LIN {X 0,Y 249.476,Z 395.408,A -85,B 0,C 180,E1 -18908.097,E2 -18908.097} C_VEL
LIN {X 0,Y 249.248,Z 395.426,A -85,B 0,C 180,E1 -18911.384,E2 -18911.384} C_VEL
LIN {X 0,Y 249.214,Z 395.443,A -85,B 0,C 180,E1 -18916.504,E2 -18916.504} C_VEL
LIN {X 0,Y 249.083,Z 395.455,A -85,B 0,C 180,E1 -18921.519,E2 -18921.519} C_VEL
LIN {X 0,Y 249.127,Z 395.443,A -85,B 0,C 180,E1 -18925.483,E2 -18925.483} C_VEL
LIN {X 0,Y 249.08,Z 395.458,A -85,B 0,C 180,E1 -18928.994,E2 -18928.994} C_VEL
LIN {X 0,Y 249.033,Z 395.457,A -85,B 0,C 180,E1 -18932.426,E2 -18932.426} C_VEL
LIN {X 0,Y 249.073,Z 395.454,A -85,B 0,C 180,E1 -18936.338,E2 -18936.338} C_VEL
LIN {X 0,Y 249.075,Z 395.455,A -85,B 0,C 180,E1 -18940.465,E2 -18940.465} C_VEL
LIN {X 0,Y 249.018,Z 395.462,A -85,B 0,C 180,E1 -18944.876,E2 -18944.876} C_VEL
LIN {X 0,Y 249.023,Z 395.464,A -85,B 0,C 180,E1 -18947.366,E2 -18947.366} C_VEL
LIN {X 0,Y 249.038,Z 395.463,A -85,B 0,C 180,E1 -18951.623,E2 -18951.623} C_VEL
LIN {X 0,Y 249.062,Z 395.462,A -85,B 0,C 180,E1 -18955.643,E2 -18955.643} C_VEL
LIN {X 0,Y 249.049,Z 395.473,A -85,B 0,C 180,E1 -18956.512,E2 -18956.512} C_VEL
LIN {X 0,Y 249.154,Z 395.988,A -85,B 0,C 180,E1 -18956.721,E2 -18956.721} C_VEL
LIN {X 0,Y 250.368,Z 398.762,A -85,B 0,C 180,E1 -18956.998,E2 -18956.998} C_VEL
LIN {X 0,Y 253.326,Z 404.095,A -85,B 0,C 180,E1 -18957.613,E2 -18957.613} C_VEL
LIN {X 0,Y 260.759,Z 419.272,A -85,B 0,C 180,E1 -18959.134,E2 -18959.134} C_VEL
LIN {X 0,Y 267.463,Z 435.997,A -85,B 0,C 180,E1 -18960.506,E2 -18960.506} C_VEL
LIN {X 0,Y 265.237,Z 502.126,A -85,B 0,C 180,E1 -18962.276,E2 -18962.276} C_VEL
LIN {X 0,Y 264.22,Z 515.294,A -85,B 0,C 180,E1 -18962.905,E2 -18962.905} C_VEL
LIN {X 0,Y 262.927,Z 527.996,A -85,B 0,C 180,E1 -18963.83,E2 -18963.83} C_VEL
LIN {X 0,Y 261.369,Z 539.299,A -85,B 0,C 180,E1 -18964.945,E2 -18964.945} C_VEL
LIN {X 0,Y 259.357,Z 550.925,A -85,B 0,C 180,E1 -18966.442,E2 -18966.442} C_VEL
LIN {X 0,Y 257.651,Z 559.929,A -85,B 0,C 180,E1 -18967.9,E2 -18967.9} C_VEL
LIN {X 0,Y 255.577,Z 569.881,A -85,B 0,C 180,E1 -18969.896,E2 -18969.896} C_VEL
LIN {X 0,Y 253.7,Z 577.735,A -85,B 0,C 180,E1 -18971.842,E2 -18971.842} C_VEL
LIN {X 0,Y 251.774,Z 585.406,A -85,B 0,C 180,E1 -18974.207,E2 -18974.207} C_VEL
LIN {X 0,Y 249.982,Z 592.445,A -85,B 0,C 180,E1 -18977.003,E2 -18977.003} C_VEL
LIN {X 0,Y 248.812,Z 597.131,A -85,B 0,C 180,E1 -18979.421,E2 -18979.421} C_VEL
LIN {X 0,Y 248.008,Z 600.712,A -85,B 0,C 180,E1 -18981.855,E2 -18981.855} C_VEL
LIN {X 0,Y 247.651,Z 602.56,A -85,B 0,C 180,E1 -18983.482,E2 -18983.482} C_VEL
LIN {X 0,Y 247.401,Z 603.948,A -85,B 0,C 180,E1 -18985.111,E2 -18985.111} C_VEL
LIN {X 0,Y 247.213,Z 604.936,A -85,B 0,C 180,E1 -18986.741,E2 -18986.741} C_VEL
LIN {X 0,Y 247.04,Z 605.774,A -85,B 0,C 180,E1 -18990,E2 -18990} C_VEL
LIN {X 0,Y 247.077,Z 605.581,A -85,B 0,C 180,E1 -18991.63,E2 -18991.63} C_VEL
LIN {X 0,Y 247.213,Z 604.996,A -85,B 0,C 180,E1 -18993.259,E2 -18993.259} C_VEL
LIN {X 0,Y 247.402,Z 604.031,A -85,B 0,C 180,E1 -18994.889,E2 -18994.889} C_VEL
LIN {X 0,Y 247.724,Z 602.386,A -85,B 0,C 180,E1 -18996.801,E2 -18996.801} C_VEL
LIN {X 0,Y 248.485,Z 598.627,A -85,B 0,C 180,E1 -18999.77,E2 -18999.77} C_VEL
LIN {X 0,Y 249.513,Z 594.382,A -85,B 0,C 180,E1 -19002.195,E2 -19002.195} C_VEL
LIN {X 0,Y 251.192,Z 587.949,A -85,B 0,C 180,E1 -19004.999,E2 -19004.999} C_VEL
LIN {X 0,Y 252.884,Z 580.88,A -85,B 0,C 180,E1 -19007.383,E2 -19007.383} C_VEL
LIN {X 0,Y 255.134,Z 572.063,A -85,B 0,C 180,E1 -19009.721,E2 -19009.721} C_VEL
LIN {X 0,Y 257.091,Z 562.672,A -85,B 0,C 180,E1 -19011.732,E2 -19011.732} C_VEL
LIN {X 0,Y 258.977,Z 552.995,A -85,B 0,C 180,E1 -19013.383,E2 -19013.383} C_VEL
LIN {X 0,Y 261.03,Z 541.835,A -85,B 0,C 180,E1 -19014.878,E2 -19014.878} C_VEL
LIN {X 0,Y 262.909,Z 529.302,A -85,B 0,C 180,E1 -19016.172,E2 -19016.172} C_VEL
LIN {X 0,Y 264.228,Z 516.356,A -85,B 0,C 180,E1 -19017.15,E2 -19017.15} C_VEL
LIN {X 0,Y 265.322,Z 503.559,A -85,B 0,C 180,E1 -19017.776,E2 -19017.776} C_VEL
LIN {X 0,Y 265.989,Z 484.214,A -85,B 0,C 180,E1 -19018.344,E2 -19018.344} C_VEL
LIN {X 0,Y 267.501,Z 436.029,A -85,B 0,C 180,E1 -19019.618,E2 -19019.618} C_VEL
LIN {X 0,Y 261.46,Z 420.884,A -85,B 0,C 180,E1 -19020.856,E2 -19020.856} C_VEL
LIN {X 0,Y 254.384,Z 406.189,A -85,B 0,C 180,E1 -19022.303,E2 -19022.303} C_VEL
LIN {X 0,Y 250.5,Z 398.916,A -85,B 0,C 180,E1 -19023.116,E2 -19023.116} C_VEL
LIN {X 0,Y 249.299,Z 396.567,A -85,B 0,C 180,E1 -19023.377,E2 -19023.377} C_VEL
LIN {X 0,Y 249.108,Z 395.797,A -85,B 0,C 180,E1 -19023.482,E2 -19023.482} C_VEL
LIN {X 0,Y 249.054,Z 395.456,A -85,B 0,C 180,E1 -19023.779,E2 -19023.779} C_VEL
LIN {X 0,Y 249.055,Z 395.462,A -85,B 0,C 180,E1 -19027.803,E2 -19027.803} C_VEL
LIN {X 0,Y 249.026,Z 395.464,A -85,B 0,C 180,E1 -19030.473,E2 -19030.473} C_VEL
LIN {X 0,Y 249.017,Z 395.465,A -85,B 0,C 180,E1 -19034.875,E2 -19034.875} C_VEL
LIN {X 0,Y 249.06,Z 395.443,A -85,B 0,C 180,E1 -19037.372,E2 -19037.372} C_VEL
LIN {X 0,Y 249.05,Z 395.46,A -85,B 0,C 180,E1 -19041.623,E2 -19041.623} C_VEL
LIN {X 0,Y 249.058,Z 395.459,A -85,B 0,C 180,E1 -19045.642,E2 -19045.642} C_VEL
LIN {X 0,Y 249.048,Z 395.464,A -85,B 0,C 180,E1 -19049.472,E2 -19049.472} C_VEL
LIN {X 0,Y 249.07,Z 395.458,A -85,B 0,C 180,E1 -19053.162,E2 -19053.162} C_VEL
LIN {X 0,Y 249.075,Z 395.451,A -85,B 0,C 180,E1 -19056.732,E2 -19056.732} C_VEL
LIN {X 0,Y 249.106,Z 395.453,A -85,B 0,C 180,E1 -19060.211,E2 -19060.211} C_VEL
LIN {X 0,Y 249.238,Z 395.433,A -85,B 0,C 180,E1 -19063.621,E2 -19063.621} C_VEL
LIN {X 0,Y 249.248,Z 395.429,A -85,B 0,C 180,E1 -19068.616,E2 -19068.616} C_VEL
LIN {X 0,Y 249.476,Z 395.408,A -85,B 0,C 180,E1 -19071.903,E2 -19071.903} C_VEL
LIN {X 0,Y 249.431,Z 395.408,A -85,B 0,C 180,E1 -19076.769,E2 -19076.769} C_VEL
LIN {X 0,Y 249.73,Z 395.374,A -85,B 0,C 180,E1 -19080,E2 -19080} C_VEL
LIN {X 0,Y 249.432,Z 395.408,A -85,B 0,C 180,E1 -19083.23,E2 -19083.23} C_VEL
LIN {X 0,Y 249.476,Z 395.399,A -85,B 0,C 180,E1 -19088.097,E2 -19088.097} C_VEL
LIN {X 0,Y 249.365,Z 395.418,A -85,B 0,C 180,E1 -19089.868,E2 -19089.868} C_VEL
LIN {X 0,Y 248.589,Z 395.52,A -85,B 0,C 180,E1 -19091.213,E2 -19091.213} C_VEL
LIN {X 0,Y 245.727,Z 395.879,A -85,B 0,C 180,E1 -19093.408,E2 -19093.408} C_VEL
LIN {X 0,Y 242.501,Z 396.283,A -85,B 0,C 180,E1 -19096.112,E2 -19096.112} C_VEL
LIN {X 0,Y 242.128,Z 396.324,A -85,B 0,C 180,E1 -19097.048,E2 -19097.048} C_VEL
LIN {X 0,Y 242.049,Z 396.333,A -85,B 0,C 180,E1 -19101.703,E2 -19101.703} C_VEL
LIN {X 0,Y 242.063,Z 396.329,A -85,B 0,C 180,E1 -19105.839,E2 -19105.839} C_VEL
LIN {X 0,Y 242.027,Z 396.335,A -85,B 0,C 180,E1 -19109.581,E2 -19109.581} C_VEL
LIN {X 0,Y 241.988,Z 396.333,A -85,B 0,C 180,E1 -19113.492,E2 -19113.492} C_VEL
LIN {X 0,Y 242.009,Z 396.332,A -85,B 0,C 180,E1 -19117.578,E2 -19117.578} C_VEL
LIN {X 0,Y 241.982,Z 396.34,A -85,B 0,C 180,E1 -19121.913,E2 -19121.913} C_VEL
LIN {X 0,Y 241.982,Z 396.34,A -85,B 0,C 180,E1 -19126.559,E2 -19126.559} C_VEL
LIN {X 0,Y 242.016,Z 396.398,A -85,B 0,C 180,E1 -19129.567,E2 -19129.567} C_VEL
LIN {X 0,Y 244.29,Z 405.347,A -85,B 0,C 180,E1 -19133.662,E2 -19133.662} C_VEL
LIN {X 0,Y 245.495,Z 411.011,A -85,B 0,C 180,E1 -19136.045,E2 -19136.045} C_VEL
LIN {X 0,Y 253.567,Z 428.776,A -85,B 0,C 180,E1 -19137.836,E2 -19137.836} C_VEL
LIN {X 0,Y 256.47,Z 436.178,A -85,B 0,C 180,E1 -19138.477,E2 -19138.477} C_VEL
LIN {X 0,Y 260.334,Z 462.518,A -85,B 0,C 180,E1 -19139.817,E2 -19139.817} C_VEL
LIN {X 0,Y 259.804,Z 485.166,A -85,B 0,C 180,E1 -19140.456,E2 -19140.456} C_VEL
LIN {X 0,Y 258.526,Z 519.992,A -85,B 0,C 180,E1 -19141.427,E2 -19141.427} C_VEL
LIN {X 0,Y 257.247,Z 533.889,A -85,B 0,C 180,E1 -19142.106,E2 -19142.106} C_VEL
LIN {X 0,Y 255.619,Z 546.328,A -85,B 0,C 180,E1 -19143.022,E2 -19143.022} C_VEL
LIN {X 0,Y 253.783,Z 557.429,A -85,B 0,C 180,E1 -19144.141,E2 -19144.141} C_VEL
LIN {X 0,Y 251.537,Z 569.003,A -85,B 0,C 180,E1 -19145.663,E2 -19145.663} C_VEL
LIN {X 0,Y 249.214,Z 579.428,A -85,B 0,C 180,E1 -19147.404,E2 -19147.404} C_VEL
LIN {X 0,Y 247.163,Z 587.956,A -85,B 0,C 180,E1 -19149.181,E2 -19149.181} C_VEL
LIN {X 0,Y 245.407,Z 596.129,A -85,B 0,C 180,E1 -19151.293,E2 -19151.293} C_VEL
LIN {X 0,Y 243.553,Z 603.536,A -85,B 0,C 180,E1 -19153.66,E2 -19153.66} C_VEL
LIN {X 0,Y 241.706,Z 610.636,A -85,B 0,C 180,E1 -19156.549,E2 -19156.549} C_VEL
LIN {X 0,Y 240.796,Z 615.372,A -85,B 0,C 180,E1 -19159.064,E2 -19159.064} C_VEL
LIN {X 0,Y 240.204,Z 618.994,A -85,B 0,C 180,E1 -19161.588,E2 -19161.588} C_VEL
LIN {X 0,Y 239.951,Z 620.862,A -85,B 0,C 180,E1 -19163.272,E2 -19163.272} C_VEL
LIN {X 0,Y 239.8,Z 622.418,A -85,B 0,C 180,E1 -19165.182,E2 -19165.182} C_VEL
LIN {X 0,Y 239.888,Z 623.885,A -85,B 0,C 180,E1 -19168.321,E2 -19168.321} C_VEL
LIN {X 0,Y 239.958,Z 624.101,A -85,B 0,C 180,E1 -19170,E2 -19170} C_VEL
LIN {X 0,Y 239.888,Z 623.875,A -85,B 0,C 180,E1 -19171.679,E2 -19171.679} C_VEL
LIN {X 0,Y 239.842,Z 622.244,A -85,B 0,C 180,E1 -19175.043,E2 -19175.043} C_VEL
LIN {X 0,Y 239.922,Z 620.829,A -85,B 0,C 180,E1 -19176.729,E2 -19176.729} C_VEL
LIN {X 0,Y 240.364,Z 617.869,A -85,B 0,C 180,E1 -19179.254,E2 -19179.254} C_VEL
LIN {X 0,Y 241.06,Z 613.867,A -85,B 0,C 180,E1 -19181.775,E2 -19181.775} C_VEL
LIN {X 0,Y 242.463,Z 607.725,A -85,B 0,C 180,E1 -19184.692,E2 -19184.692} C_VEL
LIN {X 0,Y 244.088,Z 601.024,A -85,B 0,C 180,E1 -19187.165,E2 -19187.165} C_VEL
LIN {X 0,Y 246.052,Z 593.06,A -85,B 0,C 180,E1 -19189.51,E2 -19189.51} C_VEL
LIN {X 0,Y 248.057,Z 584.199,A -85,B 0,C 180,E1 -19191.611,E2 -19191.611} C_VEL
LIN {X 0,Y 250.51,Z 573.689,A -85,B 0,C 180,E1 -19193.564,E2 -19193.564} C_VEL
LIN {X 0,Y 252.906,Z 561.859,A -85,B 0,C 180,E1 -19195.293,E2 -19195.293} C_VEL
LIN {X 0,Y 254.97,Z 549.944,A -85,B 0,C 180,E1 -19196.609,E2 -19196.609} C_VEL
LIN {X 0,Y 256.694,Z 537.544,A -85,B 0,C 180,E1 -19197.627,E2 -19197.627} C_VEL
LIN {X 0,Y 258.057,Z 524.771,A -85,B 0,C 180,E1 -19198.352,E2 -19198.352} C_VEL
LIN {X 0,Y 258.828,Z 511.246,A -85,B 0,C 180,E1 -19198.813,E2 -19198.813} C_VEL
LIN {X 0,Y 260.387,Z 463.573,A -85,B 0,C 180,E1 -19200.101,E2 -19200.101} C_VEL
LIN {X 0,Y 256.436,Z 436.34,A -85,B 0,C 180,E1 -19201.477,E2 -19201.477} C_VEL
LIN {X 0,Y 252.323,Z 425.825,A -85,B 0,C 180,E1 -19202.39,E2 -19202.39} C_VEL
LIN {X 0,Y 246.241,Z 412.845,A -85,B 0,C 180,E1 -19203.725,E2 -19203.725} C_VEL
LIN {X 0,Y 245.462,Z 410.826,A -85,B 0,C 180,E1 -19203.941,E2 -19203.941} C_VEL
LIN {X 0,Y 243.561,Z 402.34,A -85,B 0,C 180,E1 -19207.623,E2 -19207.623} C_VEL
LIN {X 0,Y 242.015,Z 396.339,A -85,B 0,C 180,E1 -19210.434,E2 -19210.434} C_VEL
LIN {X 0,Y 241.971,Z 396.331,A -85,B 0,C 180,E1 -19214.191,E2 -19214.191} C_VEL
LIN {X 0,Y 241.982,Z 396.341,A -85,B 0,C 180,E1 -19218.087,E2 -19218.087} C_VEL
LIN {X 0,Y 242.009,Z 396.335,A -85,B 0,C 180,E1 -19222.422,E2 -19222.422} C_VEL
LIN {X 0,Y 241.988,Z 396.335,A -85,B 0,C 180,E1 -19226.508,E2 -19226.508} C_VEL
LIN {X 0,Y 242.033,Z 396.33,A -85,B 0,C 180,E1 -19230.587,E2 -19230.587} C_VEL
LIN {X 0,Y 242.064,Z 396.329,A -85,B 0,C 180,E1 -19234.183,E2 -19234.183} C_VEL
LIN {X 0,Y 242.049,Z 396.329,A -85,B 0,C 180,E1 -19238.297,E2 -19238.297} C_VEL
LIN {X 0,Y 242.159,Z 396.309,A -85,B 0,C 180,E1 -19243.278,E2 -19243.278} C_VEL
LIN {X 0,Y 242.181,Z 396.313,A -85,B 0,C 180,E1 -19248.28,E2 -19248.28} C_VEL
LIN {X 0,Y 242.423,Z 396.285,A -85,B 0,C 180,E1 -19251.665,E2 -19251.665} C_VEL
LIN {X 0,Y 242.256,Z 396.304,A -85,B 0,C 180,E1 -19255.007,E2 -19255.007} C_VEL
LIN {X 0,Y 242.632,Z 396.251,A -85,B 0,C 180,E1 -19258.34,E2 -19258.34} C_VEL
LIN {X 0,Y 242.632,Z 396.26,A -85,B 0,C 180,E1 -19261.66,E2 -19261.66} C_VEL
LIN {X 0,Y 242.422,Z 396.281,A -85,B 0,C 180,E1 -19266.755,E2 -19266.755} C_VEL
LIN {X 0,Y 242.31,Z 396.299,A -85,B 0,C 180,E1 -19270.022,E2 -19270.022} C_VEL
LIN {X 0,Y 242.159,Z 396.321,A -85,B 0,C 180,E1 -19275.141,E2 -19275.141} C_VEL
LIN {X 0,Y 242.068,Z 396.321,A -85,B 0,C 180,E1 -19278.625,E2 -19278.625} C_VEL
LIN {X 0,Y 242.009,Z 396.338,A -85,B 0,C 180,E1 -19282.181,E2 -19282.181} C_VEL
LIN {X 0,Y 242.063,Z 396.321,A -85,B 0,C 180,E1 -19285.839,E2 -19285.839} C_VEL
LIN {X 0,Y 242.027,Z 396.336,A -85,B 0,C 180,E1 -19289.581,E2 -19289.581} C_VEL
LIN {X 0,Y 241.988,Z 396.34,A -85,B 0,C 180,E1 -19293.492,E2 -19293.492} C_VEL
LIN {X 0,Y 242.01,Z 396.334,A -85,B 0,C 180,E1 -19297.578,E2 -19297.578} C_VEL
LIN {X 0,Y 241.983,Z 396.338,A -85,B 0,C 180,E1 -19301.913,E2 -19301.913} C_VEL
LIN {X 0,Y 241.941,Z 396.345,A -85,B 0,C 180,E1 -19305.802,E2 -19305.802} C_VEL
LIN {X 0,Y 241.972,Z 396.344,A -85,B 0,C 180,E1 -19310.285,E2 -19310.285} C_VEL
LIN {X 0,Y 242.036,Z 396.34,A -85,B 0,C 180,E1 -19314.498,E2 -19314.498} C_VEL
LIN {X 0,Y 242.04,Z 396.336,A -85,B 0,C 180,E1 -19315.567,E2 -19315.567} C_VEL
LIN {X 0,Y 243.044,Z 399.221,A -85,B 0,C 180,E1 -19315.873,E2 -19315.873} C_VEL
LIN {X 0,Y 244.567,Z 401.612,A -85,B 0,C 180,E1 -19316.2,E2 -19316.2} C_VEL
LIN {X 0,Y 248.946,Z 409.674,A -85,B 0,C 180,E1 -19317.152,E2 -19317.152} C_VEL
LIN {X 0,Y 256.463,Z 425.531,A -85,B 0,C 180,E1 -19318.754,E2 -19318.754} C_VEL
LIN {X 0,Y 261.273,Z 437.838,A -85,B 0,C 180,E1 -19319.784,E2 -19319.784} C_VEL
LIN {X 0,Y 259.019,Z 501.868,A -85,B 0,C 180,E1 -19321.526,E2 -19321.526} C_VEL
LIN {X 0,Y 258.034,Z 514.926,A -85,B 0,C 180,E1 -19322.153,E2 -19322.153} C_VEL
LIN {X 0,Y 256.595,Z 528.27,A -85,B 0,C 180,E1 -19323.133,E2 -19323.133} C_VEL
LIN {X 0,Y 254.954,Z 539.572,A -85,B 0,C 180,E1 -19324.269,E2 -19324.269} C_VEL
LIN {X 0,Y 252.876,Z 551.196,A -85,B 0,C 180,E1 -19325.8,E2 -19325.8} C_VEL
LIN {X 0,Y 250.827,Z 561.583,A -85,B 0,C 180,E1 -19327.548,E2 -19327.548} C_VEL
LIN {X 0,Y 248.929,Z 570.151,A -85,B 0,C 180,E1 -19329.335,E2 -19329.335} C_VEL
LIN {X 0,Y 246.983,Z 578.004,A -85,B 0,C 180,E1 -19331.33,E2 -19331.33} C_VEL
LIN {X 0,Y 244.938,Z 585.675,A -85,B 0,C 180,E1 -19333.755,E2 -19333.755} C_VEL
LIN {X 0,Y 243.069,Z 592.714,A -85,B 0,C 180,E1 -19336.626,E2 -19336.626} C_VEL
LIN {X 0,Y 241.844,Z 597.399,A -85,B 0,C 180,E1 -19339.112,E2 -19339.112} C_VEL
LIN {X 0,Y 240.976,Z 600.98,A -85,B 0,C 180,E1 -19341.615,E2 -19341.615} C_VEL
LIN {X 0,Y 240.601,Z 602.828,A -85,B 0,C 180,E1 -19343.29,E2 -19343.29} C_VEL
LIN {X 0,Y 240.322,Z 604.216,A -85,B 0,C 180,E1 -19344.967,E2 -19344.967} C_VEL
LIN {X 0,Y 240.135,Z 605.203,A -85,B 0,C 180,E1 -19346.644,E2 -19346.644} C_VEL
LIN {X 0,Y 239.97,Z 606.04,A -85,B 0,C 180,E1 -19350,E2 -19350} C_VEL
LIN {X 0,Y 240.01,Z 605.847,A -85,B 0,C 180,E1 -19351.678,E2 -19351.678} C_VEL
LIN {X 0,Y 240.135,Z 605.262,A -85,B 0,C 180,E1 -19353.356,E2 -19353.356} C_VEL
LIN {X 0,Y 240.601,Z 602.945,A -85,B 0,C 180,E1 -19356.71,E2 -19356.71} C_VEL
LIN {X 0,Y 241.256,Z 600.084,A -85,B 0,C 180,E1 -19359.219,E2 -19359.219} C_VEL
LIN {X 0,Y 242.176,Z 596.204,A -85,B 0,C 180,E1 -19361.72,E2 -19361.72} C_VEL
LIN {X 0,Y 243.505,Z 591.193,A -85,B 0,C 180,E1 -19364.201,E2 -19364.201} C_VEL
LIN {X 0,Y 245.132,Z 584.882,A -85,B 0,C 180,E1 -19366.66,E2 -19366.66} C_VEL
LIN {X 0,Y 247.296,Z 576.974,A -85,B 0,C 180,E1 -19369.076,E2 -19369.076} C_VEL
LIN {X 0,Y 249.265,Z 568.914,A -85,B 0,C 180,E1 -19371.068,E2 -19371.068} C_VEL
LIN {X 0,Y 251.291,Z 559.083,A -85,B 0,C 180,E1 -19373.05,E2 -19373.05} C_VEL
LIN {X 0,Y 253.509,Z 548.002,A -85,B 0,C 180,E1 -19374.79,E2 -19374.79} C_VEL
LIN {X 0,Y 255.44,Z 537.132,A -85,B 0,C 180,E1 -19376.117,E2 -19376.117} C_VEL
LIN {X 0,Y 257.092,Z 525.12,A -85,B 0,C 180,E1 -19377.25,E2 -19377.25} C_VEL
LIN {X 0,Y 258.371,Z 512.757,A -85,B 0,C 180,E1 -19378.093,E2 -19378.093} C_VEL
LIN {X 0,Y 259.221,Z 499.909,A -85,B 0,C 180,E1 -19378.655,E2 -19378.655} C_VEL
LIN {X 0,Y 261.323,Z 437.744,A -85,B 0,C 180,E1 -19380.345,E2 -19380.345} C_VEL
LIN {X 0,Y 255.173,Z 422.628,A -85,B 0,C 180,E1 -19381.655,E2 -19381.655} C_VEL
LIN {X 0,Y 247.567,Z 406.884,A -85,B 0,C 180,E1 -19383.292,E2 -19383.292} C_VEL
LIN {X 0,Y 243.555,Z 399.903,A -85,B 0,C 180,E1 -19384.164,E2 -19384.164} C_VEL
LIN {X 0,Y 242.217,Z 397.34,A -85,B 0,C 180,E1 -19384.471,E2 -19384.471} C_VEL
LIN {X 0,Y 242.035,Z 396.333,A -85,B 0,C 180,E1 -19384.561,E2 -19384.561} C_VEL
LIN {X 0,Y 242.007,Z 396.339,A -85,B 0,C 180,E1 -19388.363,E2 -19388.363} C_VEL
LIN {X 0,Y 241.947,Z 396.347,A -85,B 0,C 180,E1 -19391.919,E2 -19391.919} C_VEL
LIN {X 0,Y 241.989,Z 396.325,A -85,B 0,C 180,E1 -19396.556,E2 -19396.556} C_VEL
LIN {X 0,Y 242.006,Z 396.34,A -85,B 0,C 180,E1 -19400.29,E2 -19400.29} C_VEL
LIN {X 0,Y 242.034,Z 396.335,A -85,B 0,C 180,E1 -19404.497,E2 -19404.497} C_VEL
LIN {X 0,Y 241.973,Z 396.343,A -85,B 0,C 180,E1 -19408.479,E2 -19408.479} C_VEL
LIN {X 0,Y 242.005,Z 396.336,A -85,B 0,C 180,E1 -19412.312,E2 -19412.312} C_VEL
LIN {X 0,Y 242.053,Z 396.326,A -85,B 0,C 180,E1 -19416.015,E2 -19416.015} C_VEL
LIN {X 0,Y 242.033,Z 396.337,A -85,B 0,C 180,E1 -19419.607,E2 -19419.607} C_VEL
LIN {X 0,Y 242.159,Z 396.312,A -85,B 0,C 180,E1 -19423.278,E2 -19423.278} C_VEL
LIN {X 0,Y 242.181,Z 396.309,A -85,B 0,C 180,E1 -19428.279,E2 -19428.279} C_VEL
LIN {X 0,Y 242.423,Z 396.288,A -85,B 0,C 180,E1 -19431.665,E2 -19431.665} C_VEL
LIN {X 0,Y 242.255,Z 396.299,A -85,B 0,C 180,E1 -19435.007,E2 -19435.007} C_VEL
LIN {X 0,Y 242.632,Z 396.26,A -85,B 0,C 180,E1 -19438.34,E2 -19438.34} C_VEL
LIN {X 0,Y 242.632,Z 396.249,A -85,B 0,C 180,E1 -19441.66,E2 -19441.66} C_VEL
LIN {X 0,Y 242.428,Z 396.285,A -85,B 0,C 180,E1 -19446.659,E2 -19446.659} C_VEL
LIN {X 0,Y 242.309,Z 396.297,A -85,B 0,C 180,E1 -19450.022,E2 -19450.022} C_VEL
LIN {X 0,Y 242.162,Z 396.314,A -85,B 0,C 180,E1 -19455.141,E2 -19455.141} C_VEL
LIN {X 0,Y 242.128,Z 396.324,A -85,B 0,C 180,E1 -19457.048,E2 -19457.048} C_VEL
LIN {X 0,Y 241.355,Z 396.419,A -85,B 0,C 180,E1 -19458.436,E2 -19458.436} C_VEL
LIN {X 0,Y 238.411,Z 396.781,A -85,B 0,C 180,E1 -19460.699,E2 -19460.699} C_VEL
LIN {X 0,Y 235.998,Z 397.089,A -85,B 0,C 180,E1 -19462.544,E2 -19462.544} C_VEL
LIN {X 0,Y 235.017,Z 397.206,A -85,B 0,C 180,E1 -19463.976,E2 -19463.976} C_VEL
LIN {X 0,Y 234.962,Z 397.21,A -85,B 0,C 180,E1 -19464.461,E2 -19464.461} C_VEL
LIN {X 0,Y 234.948,Z 397.218,A -85,B 0,C 180,E1 -19468.595,E2 -19468.595} C_VEL
LIN {X 0,Y 234.946,Z 397.21,A -85,B 0,C 180,E1 -19473.118,E2 -19473.118} C_VEL
LIN {X 0,Y 234.943,Z 397.211,A -85,B 0,C 180,E1 -19476.746,E2 -19476.746} C_VEL
LIN {X 0,Y 234.942,Z 397.215,A -85,B 0,C 180,E1 -19481.155,E2 -19481.155} C_VEL
LIN {X 0,Y 234.938,Z 397.215,A -85,B 0,C 180,E1 -19484.116,E2 -19484.116} C_VEL
LIN {X 0,Y 234.935,Z 397.218,A -85,B 0,C 180,E1 -19488.406,E2 -19488.406} C_VEL
LIN {X 0,Y 234.96,Z 397.503,A -85,B 0,C 180,E1 -19488.722,E2 -19488.722} C_VEL
LIN {X 0,Y 237.003,Z 405.178,A -85,B 0,C 180,E1 -19492.421,E2 -19492.421} C_VEL
LIN {X 0,Y 238.278,Z 410.734,A -85,B 0,C 180,E1 -19494.869,E2 -19494.869} C_VEL
LIN {X 0,Y 247.21,Z 430.033,A -85,B 0,C 180,E1 -19496.956,E2 -19496.956} C_VEL
LIN {X 0,Y 250.691,Z 438.946,A -85,B 0,C 180,E1 -19497.763,E2 -19497.763} C_VEL
LIN {X 0,Y 254.252,Z 464.097,A -85,B 0,C 180,E1 -19499.075,E2 -19499.075} C_VEL
LIN {X 0,Y 252.326,Z 519.739,A -85,B 0,C 180,E1 -19500.658,E2 -19500.658} C_VEL
LIN {X 0,Y 250.995,Z 533.631,A -85,B 0,C 180,E1 -19501.347,E2 -19501.347} C_VEL
LIN {X 0,Y 249.303,Z 546.066,A -85,B 0,C 180,E1 -19502.281,E2 -19502.281} C_VEL
LIN {X 0,Y 247.413,Z 557.166,A -85,B 0,C 180,E1 -19503.424,E2 -19503.424} C_VEL
LIN {X 0,Y 245.075,Z 568.739,A -85,B 0,C 180,E1 -19504.977,E2 -19504.977} C_VEL
LIN {X 0,Y 242.664,Z 579.164,A -85,B 0,C 180,E1 -19506.759,E2 -19506.759} C_VEL
LIN {X 0,Y 240.515,Z 587.691,A -85,B 0,C 180,E1 -19508.577,E2 -19508.577} C_VEL
LIN {X 0,Y 238.739,Z 595.369,A -85,B 0,C 180,E1 -19510.598,E2 -19510.598} C_VEL
LIN {X 0,Y 236.685,Z 603.268,A -85,B 0,C 180,E1 -19513.172,E2 -19513.172} C_VEL
LIN {X 0,Y 234.781,Z 610.369,A -85,B 0,C 180,E1 -19516.145,E2 -19516.145} C_VEL
LIN {X 0,Y 233.787,Z 615.104,A -85,B 0,C 180,E1 -19518.732,E2 -19518.732} C_VEL
LIN {X 0,Y 233.145,Z 618.726,A -85,B 0,C 180,E1 -19521.331,E2 -19521.331} C_VEL
LIN {X 0,Y 232.888,Z 620.595,A -85,B 0,C 180,E1 -19523.067,E2 -19523.067} C_VEL
LIN {X 0,Y 232.703,Z 622.334,A -85,B 0,C 180,E1 -19525.313,E2 -19525.313} C_VEL
LIN {X 0,Y 232.797,Z 623.618,A -85,B 0,C 180,E1 -19528.27,E2 -19528.27} C_VEL
LIN {X 0,Y 232.888,Z 623.835,A -85,B 0,C 180,E1 -19530,E2 -19530} C_VEL
LIN {X 0,Y 232.797,Z 623.607,A -85,B 0,C 180,E1 -19531.73,E2 -19531.73} C_VEL
LIN {X 0,Y 232.744,Z 621.976,A -85,B 0,C 180,E1 -19535.197,E2 -19535.197} C_VEL
LIN {X 0,Y 232.867,Z 620.561,A -85,B 0,C 180,E1 -19536.934,E2 -19536.934} C_VEL
LIN {X 0,Y 233.312,Z 617.599,A -85,B 0,C 180,E1 -19539.536,E2 -19539.536} C_VEL
LIN {X 0,Y 234.079,Z 613.597,A -85,B 0,C 180,E1 -19542.132,E2 -19542.132} C_VEL
LIN {X 0,Y 235.552,Z 607.455,A -85,B 0,C 180,E1 -19545.133,E2 -19545.133} C_VEL
LIN {X 0,Y 237.294,Z 600.754,A -85,B 0,C 180,E1 -19547.672,E2 -19547.672} C_VEL
LIN {X 0,Y 239.167,Z 593.466,A -85,B 0,C 180,E1 -19549.893,E2 -19549.893} C_VEL
LIN {X 0,Y 241.442,Z 583.928,A -85,B 0,C 180,E1 -19552.235,E2 -19552.235} C_VEL
LIN {X 0,Y 243.99,Z 573.418,A -85,B 0,C 180,E1 -19554.233,E2 -19554.233} C_VEL
LIN {X 0,Y 246.207,Z 563.018,A -85,B 0,C 180,E1 -19555.804,E2 -19555.804} C_VEL
LIN {X 0,Y 248.315,Z 551.613,A -85,B 0,C 180,E1 -19557.153,E2 -19557.153} C_VEL
LIN {X 0,Y 250.085,Z 539.873,A -85,B 0,C 180,E1 -19558.194,E2 -19558.194} C_VEL
LIN {X 0,Y 251.63,Z 526.548,A -85,B 0,C 180,E1 -19559.017,E2 -19559.017} C_VEL
LIN {X 0,Y 252.545,Z 513.512,A -85,B 0,C 180,E1 -19559.518,E2 -19559.518} C_VEL
LIN {X 0,Y 254.225,Z 464.328,A -85,B 0,C 180,E1 -19560.876,E2 -19560.876} C_VEL
LIN {X 0,Y 250.494,Z 438.21,A -85,B 0,C 180,E1 -19562.242,E2 -19562.242} C_VEL
LIN {X 0,Y 244.956,Z 425.063,A -85,B 0,C 180,E1 -19563.504,E2 -19563.504} C_VEL
LIN {X 0,Y 238.248,Z 410.481,A -85,B 0,C 180,E1 -19565.126,E2 -19565.126} C_VEL
LIN {X 0,Y 236.416,Z 402.809,A -85,B 0,C 180,E1 -19568.628,E2 -19568.628} C_VEL
LIN {X 0,Y 234.918,Z 397.22,A -85,B 0,C 180,E1 -19571.448,E2 -19571.448} C_VEL
LIN {X 0,Y 234.934,Z 397.207,A -85,B 0,C 180,E1 -19574.114,E2 -19574.114} C_VEL
LIN {X 0,Y 234.957,Z 397.215,A -85,B 0,C 180,E1 -19578.398,E2 -19578.398} C_VEL
LIN {X 0,Y 234.952,Z 397.219,A -85,B 0,C 180,E1 -19581.085,E2 -19581.085} C_VEL
LIN {X 0,Y 234.957,Z 397.216,A -85,B 0,C 180,E1 -19585.366,E2 -19585.366} C_VEL
LIN {X 0,Y 234.966,Z 397.211,A -85,B 0,C 180,E1 -19590.157,E2 -19590.157} C_VEL
LIN {X 0,Y 234.991,Z 397.211,A -85,B 0,C 180,E1 -19593.793,E2 -19593.793} C_VEL
LIN {X 0,Y 235.007,Z 397.208,A -85,B 0,C 180,E1 -19598.969,E2 -19598.969} C_VEL
LIN {X 0,Y 235.092,Z 397.188,A -85,B 0,C 180,E1 -19603.059,E2 -19603.059} C_VEL
LIN {X 0,Y 235.113,Z 397.193,A -85,B 0,C 180,E1 -19607.922,E2 -19607.922} C_VEL
LIN {X 0,Y 235.372,Z 397.16,A -85,B 0,C 180,E1 -19611.414,E2 -19611.414} C_VEL
LIN {X 0,Y 235.399,Z 397.165,A -85,B 0,C 180,E1 -19613.141,E2 -19613.141} C_VEL
LIN {X 0,Y 235.591,Z 397.128,A -85,B 0,C 180,E1 -19618.291,E2 -19618.291} C_VEL
LIN {X 0,Y 235.591,Z 397.137,A -85,B 0,C 180,E1 -19621.71,E2 -19621.71} C_VEL
LIN {X 0,Y 235.399,Z 397.157,A -85,B 0,C 180,E1 -19626.859,E2 -19626.859} C_VEL
LIN {X 0,Y 235.234,Z 397.179,A -85,B 0,C 180,E1 -19630.327,E2 -19630.327} C_VEL
LIN {X 0,Y 235.108,Z 397.198,A -85,B 0,C 180,E1 -19635.607,E2 -19635.607} C_VEL
LIN {X 0,Y 235.004,Z 397.197,A -85,B 0,C 180,E1 -19639.206,E2 -19639.206} C_VEL
LIN {X 0,Y 234.957,Z 397.218,A -85,B 0,C 180,E1 -19642.883,E2 -19642.883} C_VEL
LIN {X 0,Y 234.966,Z 397.207,A -85,B 0,C 180,E1 -19646.658,E2 -19646.658} C_VEL
LIN {X 0,Y 234.929,Z 397.215,A -85,B 0,C 180,E1 -19650.568,E2 -19650.568} C_VEL
LIN {X 0,Y 234.958,Z 397.218,A -85,B 0,C 180,E1 -19654.634,E2 -19654.634} C_VEL
LIN {X 0,Y 234.965,Z 397.217,A -85,B 0,C 180,E1 -19658.953,E2 -19658.953} C_VEL
LIN {X 0,Y 234.963,Z 397.216,A -85,B 0,C 180,E1 -19663.469,E2 -19663.469} C_VEL
LIN {X 0,Y 234.921,Z 397.224,A -85,B 0,C 180,E1 -19666.523,E2 -19666.523} C_VEL
LIN {X 0,Y 234.954,Z 397.216,A -85,B 0,C 180,E1 -19671.087,E2 -19671.087} C_VEL
LIN {X 0,Y 235.013,Z 397.215,A -85,B 0,C 180,E1 -19674.425,E2 -19674.425} C_VEL
LIN {X 0,Y 236.113,Z 400.261,A -85,B 0,C 180,E1 -19674.751,E2 -19674.751} C_VEL
LIN {X 0,Y 237.479,Z 402.266,A -85,B 0,C 180,E1 -19675.059,E2 -19675.059} C_VEL
LIN {X 0,Y 242.907,Z 411.835,A -85,B 0,C 180,E1 -19676.293,E2 -19676.293} C_VEL
LIN {X 0,Y 250.151,Z 427.078,A -85,B 0,C 180,E1 -19677.914,E2 -19677.914} C_VEL
LIN {X 0,Y 255.067,Z 439.434,A -85,B 0,C 180,E1 -19679.011,E2 -19679.011} C_VEL
LIN {X 0,Y 254.065,Z 468.718,A -85,B 0,C 180,E1 -19679.819,E2 -19679.819} C_VEL
LIN {X 0,Y 252.777,Z 502.806,A -85,B 0,C 180,E1 -19680.787,E2 -19680.787} C_VEL
LIN {X 0,Y 251.689,Z 516.022,A -85,B 0,C 180,E1 -19681.449,E2 -19681.449} C_VEL
LIN {X 0,Y 250.31,Z 528.543,A -85,B 0,C 180,E1 -19682.402,E2 -19682.402} C_VEL
LIN {X 0,Y 248.592,Z 539.844,A -85,B 0,C 180,E1 -19683.56,E2 -19683.56} C_VEL
LIN {X 0,Y 246.425,Z 551.467,A -85,B 0,C 180,E1 -19685.124,E2 -19685.124} C_VEL
LIN {X 0,Y 244.56,Z 560.439,A -85,B 0,C 180,E1 -19686.642,E2 -19686.642} C_VEL
LIN {X 0,Y 242.308,Z 570.421,A -85,B 0,C 180,E1 -19688.743,E2 -19688.743} C_VEL
LIN {X 0,Y 240.281,Z 578.273,A -85,B 0,C 180,E1 -19690.789,E2 -19690.789} C_VEL
LIN {X 0,Y 238.126,Z 585.945,A -85,B 0,C 180,E1 -19693.277,E2 -19693.277} C_VEL
LIN {X 0,Y 236.173,Z 592.983,A -85,B 0,C 180,E1 -19696.228,E2 -19696.228} C_VEL
LIN {X 0,Y 234.867,Z 597.667,A -85,B 0,C 180,E1 -19698.785,E2 -19698.785} C_VEL
LIN {X 0,Y 233.946,Z 601.248,A -85,B 0,C 180,E1 -19701.361,E2 -19701.361} C_VEL
LIN {X 0,Y 233.491,Z 603.336,A -85,B 0,C 180,E1 -19703.361,E2 -19703.361} C_VEL
LIN {X 0,Y 233.058,Z 605.471,A -85,B 0,C 180,E1 -19706.542,E2 -19706.542} C_VEL
LIN {X 0,Y 232.945,Z 606.077,A -85,B 0,C 180,E1 -19708.271,E2 -19708.271} C_VEL
LIN {X 0,Y 232.901,Z 606.306,A -85,B 0,C 180,E1 -19710,E2 -19710} C_VEL
LIN {X 0,Y 232.945,Z 606.113,A -85,B 0,C 180,E1 -19711.729,E2 -19711.729} C_VEL
LIN {X 0,Y 233.058,Z 605.529,A -85,B 0,C 180,E1 -19713.458,E2 -19713.458} C_VEL
LIN {X 0,Y 233.545,Z 603.211,A -85,B 0,C 180,E1 -19716.913,E2 -19716.913} C_VEL
LIN {X 0,Y 234.236,Z 600.351,A -85,B 0,C 180,E1 -19719.498,E2 -19719.498} C_VEL
LIN {X 0,Y 235.239,Z 596.47,A -85,B 0,C 180,E1 -19722.071,E2 -19722.071} C_VEL
LIN {X 0,Y 236.63,Z 591.459,A -85,B 0,C 180,E1 -19724.622,E2 -19724.622} C_VEL
LIN {X 0,Y 238.334,Z 585.147,A -85,B 0,C 180,E1 -19727.15,E2 -19727.15} C_VEL
LIN {X 0,Y 240.593,Z 577.238,A -85,B 0,C 180,E1 -19729.628,E2 -19729.628} C_VEL
LIN {X 0,Y 242.652,Z 569.178,A -85,B 0,C 180,E1 -19731.671,E2 -19731.671} C_VEL
LIN {X 0,Y 244.764,Z 559.347,A -85,B 0,C 180,E1 -19733.702,E2 -19733.702} C_VEL
LIN {X 0,Y 247.101,Z 548.264,A -85,B 0,C 180,E1 -19735.479,E2 -19735.479} C_VEL
LIN {X 0,Y 249.104,Z 537.393,A -85,B 0,C 180,E1 -19736.833,E2 -19736.833} C_VEL
LIN {X 0,Y 250.806,Z 525.379,A -85,B 0,C 180,E1 -19737.992,E2 -19737.992} C_VEL
LIN {X 0,Y 252.147,Z 513.013,A -85,B 0,C 180,E1 -19738.851,E2 -19738.851} C_VEL
LIN {X 0,Y 253.033,Z 500.159,A -85,B 0,C 180,E1 -19739.423,E2 -19739.423} C_VEL
LIN {X 0,Y 255.182,Z 439.559,A -85,B 0,C 180,E1 -19741.105,E2 -19741.105} C_VEL
LIN {X 0,Y 249.579,Z 425.803,A -85,B 0,C 180,E1 -19742.351,E2 -19742.351} C_VEL
LIN {X 0,Y 242.543,Z 411.061,A -85,B 0,C 180,E1 -19743.935,E2 -19743.935} C_VEL
LIN {X 0,Y 236.521,Z 400.814,A -85,B 0,C 180,E1 -19745.306,E2 -19745.306} C_VEL
LIN {X 0,Y 235.154,Z 398.128,A -85,B 0,C 180,E1 -19745.643,E2 -19745.643} C_VEL
LIN {X 0,Y 234.981,Z 397.216,A -85,B 0,C 180,E1 -19745.72,E2 -19745.72} C_VEL
LIN {X 0,Y 234.941,Z 397.22,A -85,B 0,C 180,E1 -19748.944,E2 -19748.944} C_VEL
LIN {X 0,Y 234.921,Z 397.22,A -85,B 0,C 180,E1 -19753.477,E2 -19753.477} C_VEL
LIN {X 0,Y 234.963,Z 397.199,A -85,B 0,C 180,E1 -19756.531,E2 -19756.531} C_VEL
LIN {X 0,Y 234.953,Z 397.219,A -85,B 0,C 180,E1 -19761.085,E2 -19761.085} C_VEL
LIN {X 0,Y 234.958,Z 397.217,A -85,B 0,C 180,E1 -19765.366,E2 -19765.366} C_VEL
LIN {X 0,Y 234.966,Z 397.213,A -85,B 0,C 180,E1 -19770.157,E2 -19770.157} C_VEL
LIN {X 0,Y 234.991,Z 397.214,A -85,B 0,C 180,E1 -19773.793,E2 -19773.793} C_VEL
LIN {X 0,Y 235.007,Z 397.21,A -85,B 0,C 180,E1 -19778.969,E2 -19778.969} C_VEL
LIN {X 0,Y 235.092,Z 397.191,A -85,B 0,C 180,E1 -19783.059,E2 -19783.059} C_VEL
LIN {X 0,Y 235.113,Z 397.19,A -85,B 0,C 180,E1 -19787.922,E2 -19787.922} C_VEL
LIN {X 0,Y 235.372,Z 397.167,A -85,B 0,C 180,E1 -19791.414,E2 -19791.414} C_VEL
LIN {X 0,Y 235.399,Z 397.162,A -85,B 0,C 180,E1 -19793.141,E2 -19793.141} C_VEL
LIN {X 0,Y 235.591,Z 397.137,A -85,B 0,C 180,E1 -19798.29,E2 -19798.29} C_VEL
LIN {X 0,Y 235.592,Z 397.125,A -85,B 0,C 180,E1 -19801.709,E2 -19801.709} C_VEL
LIN {X 0,Y 235.399,Z 397.158,A -85,B 0,C 180,E1 -19806.859,E2 -19806.859} C_VEL
LIN {X 0,Y 235.234,Z 397.179,A -85,B 0,C 180,E1 -19810.327,E2 -19810.327} C_VEL
LIN {X 0,Y 235.109,Z 397.195,A -85,B 0,C 180,E1 -19815.607,E2 -19815.607} C_VEL
LIN {X 0,Y 235.004,Z 397.203,A -85,B 0,C 180,E1 -19819.206,E2 -19819.206} C_VEL
LIN {X 0,Y 234.957,Z 397.217,A -85,B 0,C 180,E1 -19822.883,E2 -19822.883} C_VEL
LIN {X 0,Y 234.962,Z 397.21,A -85,B 0,C 180,E1 -19824.461,E2 -19824.461} C_VEL
LIN {X 0,Y 234.356,Z 397.29,A -85,B 0,C 180,E1 -19825.892,E2 -19825.892} C_VEL
LIN {X 0,Y 232.791,Z 397.49,A -85,B 0,C 180,E1 -19827.297,E2 -19827.297} C_VEL
LIN {X 0,Y 229.026,Z 397.96,A -85,B 0,C 180,E1 -19830.128,E2 -19830.128} C_VEL
LIN {X 0,Y 227.944,Z 398.089,A -85,B 0,C 180,E1 -19831.606,E2 -19831.606} C_VEL
LIN {X 0,Y 227.848,Z 398.096,A -85,B 0,C 180,E1 -19832.108,E2 -19832.108} C_VEL
LIN {X 0,Y 227.906,Z 398.088,A -85,B 0,C 180,E1 -19836.702,E2 -19836.702} C_VEL
LIN {X 0,Y 227.89,Z 398.091,A -85,B 0,C 180,E1 -19840.363,E2 -19840.363} C_VEL
LIN {X 0,Y 227.907,Z 398.091,A -85,B 0,C 180,E1 -19842.72,E2 -19842.72} C_VEL
LIN {X 0,Y 227.883,Z 398.197,A -85,B 0,C 180,E1 -19847.625,E2 -19847.625} C_VEL
LIN {X 0,Y 230.184,Z 406.96,A -85,B 0,C 180,E1 -19852.024,E2 -19852.024} C_VEL
LIN {X 0,Y 230.966,Z 410.19,A -85,B 0,C 180,E1 -19853.558,E2 -19853.558} C_VEL
LIN {X 0,Y 240.745,Z 431.061,A -85,B 0,C 180,E1 -19855.995,E2 -19855.995} C_VEL
LIN {X 0,Y 244.902,Z 441.495,A -85,B 0,C 180,E1 -19857,E2 -19857} C_VEL
LIN {X 0,Y 248.165,Z 465.164,A -85,B 0,C 180,E1 -19858.273,E2 -19858.273} C_VEL
LIN {X 0,Y 246.231,Z 518.855,A -85,B 0,C 180,E1 -19859.825,E2 -19859.825} C_VEL
LIN {X 0,Y 244.982,Z 531.951,A -85,B 0,C 180,E1 -19860.466,E2 -19860.466} C_VEL
LIN {X 0,Y 243.216,Z 544.696,A -85,B 0,C 180,E1 -19861.407,E2 -19861.407} C_VEL
LIN {X 0,Y 241.065,Z 556.903,A -85,B 0,C 180,E1 -19862.667,E2 -19862.667} C_VEL
LIN {X 0,Y 238.646,Z 568.475,A -85,B 0,C 180,E1 -19864.255,E2 -19864.255} C_VEL
LIN {X 0,Y 236.127,Z 578.899,A -85,B 0,C 180,E1 -19866.076,E2 -19866.076} C_VEL
LIN {X 0,Y 233.897,Z 587.425,A -85,B 0,C 180,E1 -19867.94,E2 -19867.94} C_VEL
LIN {X 0,Y 232.017,Z 594.693,A -85,B 0,C 180,E1 -19869.887,E2 -19869.887} C_VEL
LIN {X 0,Y 230.152,Z 601.841,A -85,B 0,C 180,E1 -19872.22,E2 -19872.22} C_VEL
LIN {X 0,Y 228.428,Z 608.279,A -85,B 0,C 180,E1 -19874.84,E2 -19874.84} C_VEL
LIN {X 0,Y 227.087,Z 613.396,A -85,B 0,C 180,E1 -19877.489,E2 -19877.489} C_VEL
LIN {X 0,Y 226.283,Z 617.38,A -85,B 0,C 180,E1 -19880.165,E2 -19880.165} C_VEL
LIN {X 0,Y 225.818,Z 620.328,A -85,B 0,C 180,E1 -19882.849,E2 -19882.849} C_VEL
LIN {X 0,Y 225.605,Z 622.255,A -85,B 0,C 180,E1 -19885.46,E2 -19885.46} C_VEL
LIN {X 0,Y 225.707,Z 623.351,A -85,B 0,C 180,E1 -19888.216,E2 -19888.216} C_VEL
LIN {X 0,Y 225.819,Z 623.569,A -85,B 0,C 180,E1 -19890,E2 -19890} C_VEL
LIN {X 0,Y 225.708,Z 623.34,A -85,B 0,C 180,E1 -19891.784,E2 -19891.784} C_VEL
LIN {X 0,Y 225.671,Z 622.101,A -85,B 0,C 180,E1 -19894.747,E2 -19894.747} C_VEL
LIN {X 0,Y 225.802,Z 620.293,A -85,B 0,C 180,E1 -19897.152,E2 -19897.152} C_VEL
LIN {X 0,Y 226.283,Z 617.33,A -85,B 0,C 180,E1 -19899.835,E2 -19899.835} C_VEL
LIN {X 0,Y 227.084,Z 613.326,A -85,B 0,C 180,E1 -19902.512,E2 -19902.512} C_VEL
LIN {X 0,Y 228.675,Z 607.185,A -85,B 0,C 180,E1 -19905.6,E2 -19905.6} C_VEL
LIN {X 0,Y 230.527,Z 600.485,A -85,B 0,C 180,E1 -19908.209,E2 -19908.209} C_VEL
LIN {X 0,Y 232.815,Z 591.83,A -85,B 0,C 180,E1 -19910.88,E2 -19910.88} C_VEL
LIN {X 0,Y 234.876,Z 583.658,A -85,B 0,C 180,E1 -19912.891,E2 -19912.891} C_VEL
LIN {X 0,Y 237.485,Z 573.145,A -85,B 0,C 180,E1 -19914.942,E2 -19914.942} C_VEL
LIN {X 0,Y 240.123,Z 561.315,A -85,B 0,C 180,E1 -19916.743,E2 -19916.743} C_VEL
LIN {X 0,Y 242.357,Z 549.398,A -85,B 0,C 180,E1 -19918.113,E2 -19918.113} C_VEL
LIN {X 0,Y 244.224,Z 536.995,A -85,B 0,C 180,E1 -19919.17,E2 -19919.17} C_VEL
LIN {X 0,Y 245.695,Z 523.858,A -85,B 0,C 180,E1 -19919.94,E2 -19919.94} C_VEL
LIN {X 0,Y 246.569,Z 509.115,A -85,B 0,C 180,E1 -19920.444,E2 -19920.444} C_VEL
LIN {X 0,Y 248.08,Z 465.032,A -85,B 0,C 180,E1 -19921.695,E2 -19921.695} C_VEL
LIN {X 0,Y 244.685,Z 440.781,A -85,B 0,C 180,E1 -19923.007,E2 -19923.007} C_VEL
LIN {X 0,Y 239.251,Z 427.869,A -85,B 0,C 180,E1 -19924.303,E2 -19924.303} C_VEL
LIN {X 0,Y 232.502,Z 413.601,A -85,B 0,C 180,E1 -19925.963,E2 -19925.963} C_VEL
LIN {X 0,Y 230.934,Z 410.105,A -85,B 0,C 180,E1 -19926.431,E2 -19926.431} C_VEL
LIN {X 0,Y 229.065,Z 402.472,A -85,B 0,C 180,E1 -19930.112,E2 -19930.112} C_VEL
LIN {X 0,Y 227.894,Z 398.095,A -85,B 0,C 180,E1 -19932.412,E2 -19932.412} C_VEL
LIN {X 0,Y 227.907,Z 398.091,A -85,B 0,C 180,E1 -19937.28,E2 -19937.28} C_VEL
LIN {X 0,Y 227.869,Z 398.098,A -85,B 0,C 180,E1 -19941.914,E2 -19941.914} C_VEL
LIN {X 0,Y 227.887,Z 398.091,A -85,B 0,C 180,E1 -19946.373,E2 -19946.373} C_VEL
LIN {X 0,Y 227.916,Z 398.088,A -85,B 0,C 180,E1 -19950.437,E2 -19950.437} C_VEL
LIN {X 0,Y 227.925,Z 398.09,A -85,B 0,C 180,E1 -19954.425,E2 -19954.425} C_VEL
LIN {X 0,Y 227.958,Z 398.084,A -85,B 0,C 180,E1 -19958.287,E2 -19958.287} C_VEL
LIN {X 0,Y 228.03,Z 398.067,A -85,B 0,C 180,E1 -19962.826,E2 -19962.826} C_VEL
LIN {X 0,Y 228.07,Z 398.072,A -85,B 0,C 180,E1 -19967.543,E2 -19967.543} C_VEL
LIN {X 0,Y 228.301,Z 398.037,A -85,B 0,C 180,E1 -19971.146,E2 -19971.146} C_VEL
LIN {X 0,Y 228.35,Z 398.041,A -85,B 0,C 180,E1 -19972.928,E2 -19972.928} C_VEL
LIN {X 0,Y 228.55,Z 398.004,A -85,B 0,C 180,E1 -19978.238,E2 -19978.238} C_VEL
LIN {X 0,Y 228.55,Z 398.014,A -85,B 0,C 180,E1 -19981.762,E2 -19981.762} C_VEL
LIN {X 0,Y 228.35,Z 398.037,A -85,B 0,C 180,E1 -19987.072,E2 -19987.072} C_VEL
LIN {X 0,Y 228.155,Z 398.057,A -85,B 0,C 180,E1 -19990.651,E2 -19990.651} C_VEL
LIN {X 0,Y 228.058,Z 398.071,A -85,B 0,C 180,E1 -19994.273,E2 -19994.273} C_VEL
LIN {X 0,Y 227.999,Z 398.079,A -85,B 0,C 180,E1 -19997.954,E2 -19997.954} C_VEL
LIN {X 0,Y 227.926,Z 398.093,A -85,B 0,C 180,E1 -20002.33,E2 -20002.33} C_VEL
LIN {X 0,Y 227.94,Z 398.081,A -85,B 0,C 180,E1 -20006.603,E2 -20006.603} C_VEL
LIN {X 0,Y 227.906,Z 398.092,A -85,B 0,C 180,E1 -20010.297,E2 -20010.297} C_VEL
LIN {X 0,Y 227.887,Z 398.097,A -85,B 0,C 180,E1 -20013.719,E2 -20013.719} C_VEL
LIN {X 0,Y 227.869,Z 398.097,A -85,B 0,C 180,E1 -20018.086,E2 -20018.086} C_VEL
LIN {X 0,Y 227.907,Z 398.097,A -85,B 0,C 180,E1 -20022.72,E2 -20022.72} C_VEL
LIN {X 0,Y 227.831,Z 398.102,A -85,B 0,C 180,E1 -20027.761,E2 -20027.761} C_VEL
LIN {X 0,Y 227.869,Z 398.102,A -85,B 0,C 180,E1 -20031.915,E2 -20031.915} C_VEL
LIN {X 0,Y 227.925,Z 398.242,A -85,B 0,C 180,E1 -20033.189,E2 -20033.189} C_VEL
LIN {X 0,Y 228.904,Z 400.93,A -85,B 0,C 180,E1 -20033.477,E2 -20033.477} C_VEL
LIN {X 0,Y 230.67,Z 403.491,A -85,B 0,C 180,E1 -20033.902,E2 -20033.902} C_VEL
LIN {X 0,Y 237.571,Z 415.411,A -85,B 0,C 180,E1 -20035.549,E2 -20035.549} C_VEL
LIN {X 0,Y 244.825,Z 430.777,A -85,B 0,C 180,E1 -20037.247,E2 -20037.247} C_VEL
LIN {X 0,Y 249.033,Z 441.412,A -85,B 0,C 180,E1 -20038.23,E2 -20038.23} C_VEL
LIN {X 0,Y 246.658,Z 502.673,A -85,B 0,C 180,E1 -20039.968,E2 -20039.968} C_VEL
LIN {X 0,Y 245.462,Z 516.388,A -85,B 0,C 180,E1 -20040.662,E2 -20040.662} C_VEL
LIN {X 0,Y 244.065,Z 528.817,A -85,B 0,C 180,E1 -20041.633,E2 -20041.633} C_VEL
LIN {X 0,Y 242.271,Z 540.116,A -85,B 0,C 180,E1 -20042.814,E2 -20042.814} C_VEL
LIN {X 0,Y 240.007,Z 551.738,A -85,B 0,C 180,E1 -20044.411,E2 -20044.411} C_VEL
LIN {X 0,Y 238.029,Z 560.869,A -85,B 0,C 180,E1 -20045.996,E2 -20045.996} C_VEL
LIN {X 0,Y 235.715,Z 570.691,A -85,B 0,C 180,E1 -20048.119,E2 -20048.119} C_VEL
LIN {X 0,Y 233.6,Z 578.542,A -85,B 0,C 180,E1 -20050.217,E2 -20050.217} C_VEL
LIN {X 0,Y 231.337,Z 586.214,A -85,B 0,C 180,E1 -20052.771,E2 -20052.771} C_VEL
LIN {X 0,Y 229.295,Z 593.251,A -85,B 0,C 180,E1 -20055.806,E2 -20055.806} C_VEL
LIN {X 0,Y 227.911,Z 597.936,A -85,B 0,C 180,E1 -20058.438,E2 -20058.438} C_VEL
LIN {X 0,Y 226.918,Z 601.517,A -85,B 0,C 180,E1 -20061.092,E2 -20061.092} C_VEL
LIN {X 0,Y 226.392,Z 603.811,A -85,B 0,C 180,E1 -20063.412,E2 -20063.412} C_VEL
LIN {X 0,Y 225.985,Z 605.738,A -85,B 0,C 180,E1 -20066.434,E2 -20066.434} C_VEL
LIN {X 0,Y 225.834,Z 606.572,A -85,B 0,C 180,E1 -20070,E2 -20070} C_VEL
LIN {X 0,Y 225.859,Z 606.379,A -85,B 0,C 180,E1 -20071.783,E2 -20071.783} C_VEL
LIN {X 0,Y 225.984,Z 605.795,A -85,B 0,C 180,E1 -20073.566,E2 -20073.566} C_VEL
LIN {X 0,Y 226.501,Z 603.478,A -85,B 0,C 180,E1 -20077.129,E2 -20077.129} C_VEL
LIN {X 0,Y 227.244,Z 600.617,A -85,B 0,C 180,E1 -20079.793,E2 -20079.793} C_VEL
LIN {X 0,Y 228.289,Z 596.736,A -85,B 0,C 180,E1 -20082.445,E2 -20082.445} C_VEL
LIN {X 0,Y 229.753,Z 591.725,A -85,B 0,C 180,E1 -20085.07,E2 -20085.07} C_VEL
LIN {X 0,Y 231.557,Z 585.412,A -85,B 0,C 180,E1 -20087.668,E2 -20087.668} C_VEL
LIN {X 0,Y 233.911,Z 577.503,A -85,B 0,C 180,E1 -20090.213,E2 -20090.213} C_VEL
LIN {X 0,Y 236.07,Z 569.442,A -85,B 0,C 180,E1 -20092.307,E2 -20092.307} C_VEL
LIN {X 0,Y 238.281,Z 559.61,A -85,B 0,C 180,E1 -20094.388,E2 -20094.388} C_VEL
LIN {X 0,Y 240.724,Z 548.525,A -85,B 0,C 180,E1 -20096.204,E2 -20096.204} C_VEL
LIN {X 0,Y 242.813,Z 537.653,A -85,B 0,C 180,E1 -20097.587,E2 -20097.587} C_VEL
LIN {X 0,Y 244.571,Z 525.638,A -85,B 0,C 180,E1 -20098.771,E2 -20098.771} C_VEL
LIN {X 0,Y 245.952,Z 513.533,A -85,B 0,C 180,E1 -20099.631,E2 -20099.631} C_VEL
LIN {X 0,Y 246.884,Z 499.983,A -85,B 0,C 180,E1 -20100.248,E2 -20100.248} C_VEL
LIN {X 0,Y 249.12,Z 441.451,A -85,B 0,C 180,E1 -20101.895,E2 -20101.895} C_VEL
LIN {X 0,Y 242.664,Z 425.852,A -85,B 0,C 180,E1 -20103.399,E2 -20103.399} C_VEL
LIN {X 0,Y 235.902,Z 412.295,A -85,B 0,C 180,E1 -20104.993,E2 -20104.993} C_VEL
LIN {X 0,Y 229.846,Z 402.159,A -85,B 0,C 180,E1 -20106.452,E2 -20106.452} C_VEL
LIN {X 0,Y 228.304,Z 399.758,A -85,B 0,C 180,E1 -20106.834,E2 -20106.834} C_VEL
LIN {X 0,Y 227.888,Z 398.1,A -85,B 0,C 180,E1 -20106.987,E2 -20106.987} C_VEL
LIN {X 0,Y 227.835,Z 398.103,A -85,B 0,C 180,E1 -20110.374,E2 -20110.374} C_VEL
LIN {X 0,Y 227.849,Z 398.103,A -85,B 0,C 180,E1 -20114.811,E2 -20114.811} C_VEL
LIN {X 0,Y 227.908,Z 398.076,A -85,B 0,C 180,E1 -20117.738,E2 -20117.738} C_VEL
LIN {X 0,Y 227.869,Z 398.095,A -85,B 0,C 180,E1 -20121.914,E2 -20121.914} C_VEL
LIN {X 0,Y 227.887,Z 398.091,A -85,B 0,C 180,E1 -20126.372,E2 -20126.372} C_VEL
LIN {X 0,Y 227.916,Z 398.091,A -85,B 0,C 180,E1 -20130.437,E2 -20130.437} C_VEL
LIN {X 0,Y 227.925,Z 398.093,A -85,B 0,C 180,E1 -20134.425,E2 -20134.425} C_VEL
LIN {X 0,Y 227.958,Z 398.087,A -85,B 0,C 180,E1 -20138.287,E2 -20138.287} C_VEL
LIN {X 0,Y 228.031,Z 398.069,A -85,B 0,C 180,E1 -20142.826,E2 -20142.826} C_VEL
LIN {X 0,Y 228.07,Z 398.069,A -85,B 0,C 180,E1 -20147.543,E2 -20147.543} C_VEL
LIN {X 0,Y 228.301,Z 398.045,A -85,B 0,C 180,E1 -20151.146,E2 -20151.146} C_VEL
LIN {X 0,Y 228.35,Z 398.042,A -85,B 0,C 180,E1 -20152.928,E2 -20152.928} C_VEL
LIN {X 0,Y 228.55,Z 398.014,A -85,B 0,C 180,E1 -20158.238,E2 -20158.238} C_VEL
LIN {X 0,Y 228.55,Z 398.001,A -85,B 0,C 180,E1 -20161.762,E2 -20161.762} C_VEL
LIN {X 0,Y 228.35,Z 398.033,A -85,B 0,C 180,E1 -20167.072,E2 -20167.072} C_VEL
LIN {X 0,Y 228.159,Z 398.062,A -85,B 0,C 180,E1 -20170.651,E2 -20170.651} C_VEL
LIN {X 0,Y 228.06,Z 398.066,A -85,B 0,C 180,E1 -20174.272,E2 -20174.272} C_VEL
LIN {X 0,Y 227.999,Z 398.082,A -85,B 0,C 180,E1 -20177.954,E2 -20177.954} C_VEL
LIN {X 0,Y 227.926,Z 398.094,A -85,B 0,C 180,E1 -20182.33,E2 -20182.33} C_VEL
LIN {X 0,Y 227.939,Z 398.092,A -85,B 0,C 180,E1 -20186.603,E2 -20186.603} C_VEL
LIN {X 0,Y 227.905,Z 398.094,A -85,B 0,C 180,E1 -20190.297,E2 -20190.297} C_VEL
LIN {X 0,Y 227.848,Z 398.096,A -85,B 0,C 180,E1 -20192.108,E2 -20192.108} C_VEL
LIN {X 0,Y 227.164,Z 398.179,A -85,B 0,C 180,E1 -20193.584,E2 -20193.584} C_VEL
LIN {X 0,Y 224.331,Z 398.537,A -85,B 0,C 180,E1 -20195.995,E2 -20195.995} C_VEL
LIN {X 0,Y 221.941,Z 398.837,A -85,B 0,C 180,E1 -20197.962,E2 -20197.962} C_VEL
LIN {X 0,Y 220.926,Z 398.961,A -85,B 0,C 180,E1 -20199.488,E2 -20199.488} C_VEL
LIN {X 0,Y 220.848,Z 398.968,A -85,B 0,C 180,E1 -20200.005,E2 -20200.005} C_VEL
LIN {X 0,Y 220.83,Z 398.974,A -85,B 0,C 180,E1 -20204.44,E2 -20204.44} C_VEL
LIN {X 0,Y 220.828,Z 399.085,A -85,B 0,C 180,E1 -20206.532,E2 -20206.532} C_VEL
LIN {X 0,Y 223.058,Z 407.416,A -85,B 0,C 180,E1 -20210.94,E2 -20210.94} C_VEL
LIN {X 0,Y 223.737,Z 410.094,A -85,B 0,C 180,E1 -20212.204,E2 -20212.204} C_VEL
LIN {X 0,Y 231.223,Z 425.414,A -85,B 0,C 180,E1 -20214.192,E2 -20214.192} C_VEL
LIN {X 0,Y 237.41,Z 439.419,A -85,B 0,C 180,E1 -20215.755,E2 -20215.755} C_VEL
LIN {X 0,Y 239.143,Z 443.988,A -85,B 0,C 180,E1 -20216.196,E2 -20216.196} C_VEL
LIN {X 0,Y 242.148,Z 466.227,A -85,B 0,C 180,E1 -20217.434,E2 -20217.434} C_VEL
LIN {X 0,Y 240.079,Z 519.147,A -85,B 0,C 180,E1 -20218.997,E2 -20218.997} C_VEL
LIN {X 0,Y 238.729,Z 532.53,A -85,B 0,C 180,E1 -20219.679,E2 -20219.679} C_VEL
LIN {X 0,Y 236.831,Z 545.545,A -85,B 0,C 180,E1 -20220.684,E2 -20220.684} C_VEL
LIN {X 0,Y 234.456,Z 558.226,A -85,B 0,C 180,E1 -20222.072,E2 -20222.072} C_VEL
LIN {X 0,Y 231.98,Z 569.508,A -85,B 0,C 180,E1 -20223.7,E2 -20223.7} C_VEL
LIN {X 0,Y 229.362,Z 579.671,A -85,B 0,C 180,E1 -20225.566,E2 -20225.566} C_VEL
LIN {X 0,Y 226.843,Z 588.833,A -85,B 0,C 180,E1 -20227.696,E2 -20227.696} C_VEL
LIN {X 0,Y 224.869,Z 596.417,A -85,B 0,C 180,E1 -20229.892,E2 -20229.892} C_VEL
LIN {X 0,Y 222.741,Z 603.858,A -85,B 0,C 180,E1 -20232.558,E2 -20232.558} C_VEL
LIN {X 0,Y 220.987,Z 609.836,A -85,B 0,C 180,E1 -20235.261,E2 -20235.261} C_VEL
LIN {X 0,Y 219.787,Z 614.568,A -85,B 0,C 180,E1 -20238.004,E2 -20238.004} C_VEL
LIN {X 0,Y 219.056,Z 618.191,A -85,B 0,C 180,E1 -20240.769,E2 -20240.769} C_VEL
LIN {X 0,Y 218.754,Z 620.06,A -85,B 0,C 180,E1 -20242.617,E2 -20242.617} C_VEL
LIN {X 0,Y 218.52,Z 622.138,A -85,B 0,C 180,E1 -20245.574,E2 -20245.574} C_VEL
LIN {X 0,Y 218.62,Z 623.084,A -85,B 0,C 180,E1 -20248.158,E2 -20248.158} C_VEL
LIN {X 0,Y 218.728,Z 623.302,A -85,B 0,C 180,E1 -20250,E2 -20250} C_VEL
LIN {X 0,Y 218.621,Z 623.073,A -85,B 0,C 180,E1 -20251.842,E2 -20251.842} C_VEL
LIN {X 0,Y 218.571,Z 621.439,A -85,B 0,C 180,E1 -20255.535,E2 -20255.535} C_VEL
LIN {X 0,Y 218.726,Z 620.024,A -85,B 0,C 180,E1 -20257.384,E2 -20257.384} C_VEL
LIN {X 0,Y 219.272,Z 617.061,A -85,B 0,C 180,E1 -20260.153,E2 -20260.153} C_VEL
LIN {X 0,Y 220.104,Z 613.056,A -85,B 0,C 180,E1 -20262.915,E2 -20262.915} C_VEL
LIN {X 0,Y 221.826,Z 606.915,A -85,B 0,C 180,E1 -20266.094,E2 -20266.094} C_VEL
LIN {X 0,Y 223.786,Z 600.216,A -85,B 0,C 180,E1 -20268.778,E2 -20268.778} C_VEL
LIN {X 0,Y 226.101,Z 591.733,A -85,B 0,C 180,E1 -20271.476,E2 -20271.476} C_VEL
LIN {X 0,Y 228.322,Z 583.387,A -85,B 0,C 180,E1 -20273.587,E2 -20273.587} C_VEL
LIN {X 0,Y 231.065,Z 572.874,A -85,B 0,C 180,E1 -20275.684,E2 -20275.684} C_VEL
LIN {X 0,Y 233.811,Z 561.043,A -85,B 0,C 180,E1 -20277.525,E2 -20277.525} C_VEL
LIN {X 0,Y 236.114,Z 549.124,A -85,B 0,C 180,E1 -20278.926,E2 -20278.926} C_VEL
LIN {X 0,Y 238.048,Z 536.72,A -85,B 0,C 180,E1 -20280.003,E2 -20280.003} C_VEL
LIN {X 0,Y 239.536,Z 523.946,A -85,B 0,C 180,E1 -20280.77,E2 -20280.77} C_VEL
LIN {X 0,Y 240.428,Z 509.939,A -85,B 0,C 180,E1 -20281.27,E2 -20281.27} C_VEL
LIN {X 0,Y 242.042,Z 466.058,A -85,B 0,C 180,E1 -20282.537,E2 -20282.537} C_VEL
LIN {X 0,Y 238.904,Z 443.222,A -85,B 0,C 180,E1 -20283.816,E2 -20283.816} C_VEL
LIN {X 0,Y 233.113,Z 429.56,A -85,B 0,C 180,E1 -20285.266,E2 -20285.266} C_VEL
LIN {X 0,Y 226.962,Z 416.675,A -85,B 0,C 180,E1 -20286.855,E2 -20286.855} C_VEL
LIN {X 0,Y 223.673,Z 409.841,A -85,B 0,C 180,E1 -20287.785,E2 -20287.785} C_VEL
LIN {X 0,Y 221.645,Z 402.124,A -85,B 0,C 180,E1 -20291.748,E2 -20291.748} C_VEL
LIN {X 0,Y 220.817,Z 398.97,A -85,B 0,C 180,E1 -20293.48,E2 -20293.48} C_VEL
LIN {X 0,Y 220.851,Z 398.974,A -85,B 0,C 180,E1 -20298.066,E2 -20298.066} C_VEL
LIN {X 0,Y 220.836,Z 398.971,A -85,B 0,C 180,E1 -20302.711,E2 -20302.711} C_VEL
LIN {X 0,Y 220.821,Z 398.971,A -85,B 0,C 180,E1 -20307.245,E2 -20307.245} C_VEL
LIN {X 0,Y 220.833,Z 398.965,A -85,B 0,C 180,E1 -20311.486,E2 -20311.486} C_VEL
LIN {X 0,Y 220.864,Z 398.963,A -85,B 0,C 180,E1 -20315.565,E2 -20315.565} C_VEL
LIN {X 0,Y 220.888,Z 398.97,A -85,B 0,C 180,E1 -20319.514,E2 -20319.514} C_VEL
LIN {X 0,Y 221.012,Z 398.941,A -85,B 0,C 180,E1 -20323.37,E2 -20323.37} C_VEL
LIN {X 0,Y 221.102,Z 398.929,A -85,B 0,C 180,E1 -20329.005,E2 -20329.005} C_VEL
LIN {X 0,Y 221.285,Z 398.919,A -85,B 0,C 180,E1 -20332.701,E2 -20332.701} C_VEL
LIN {X 0,Y 221.508,Z 398.881,A -85,B 0,C 180,E1 -20338.182,E2 -20338.182} C_VEL
LIN {X 0,Y 221.508,Z 398.891,A -85,B 0,C 180,E1 -20341.818,E2 -20341.818} C_VEL
LIN {X 0,Y 221.301,Z 398.917,A -85,B 0,C 180,E1 -20347.298,E2 -20347.298} C_VEL
LIN {X 0,Y 221.102,Z 398.932,A -85,B 0,C 180,E1 -20350.995,E2 -20350.995} C_VEL
LIN {X 0,Y 221.012,Z 398.955,A -85,B 0,C 180,E1 -20356.63,E2 -20356.63} C_VEL
LIN {X 0,Y 220.888,Z 398.958,A -85,B 0,C 180,E1 -20360.487,E2 -20360.487} C_VEL
LIN {X 0,Y 220.864,Z 398.967,A -85,B 0,C 180,E1 -20364.436,E2 -20364.436} C_VEL
LIN {X 0,Y 220.834,Z 398.977,A -85,B 0,C 180,E1 -20368.514,E2 -20368.514} C_VEL
LIN {X 0,Y 220.822,Z 398.971,A -85,B 0,C 180,E1 -20372.756,E2 -20372.756} C_VEL
LIN {X 0,Y 220.836,Z 398.969,A -85,B 0,C 180,E1 -20377.289,E2 -20377.289} C_VEL
LIN {X 0,Y 220.851,Z 398.97,A -85,B 0,C 180,E1 -20381.934,E2 -20381.934} C_VEL
LIN {X 0,Y 220.788,Z 398.979,A -85,B 0,C 180,E1 -20385.551,E2 -20385.551} C_VEL
LIN {X 0,Y 220.809,Z 398.978,A -85,B 0,C 180,E1 -20390.465,E2 -20390.465} C_VEL
LIN {X 0,Y 220.843,Z 398.976,A -85,B 0,C 180,E1 -20391.793,E2 -20391.793} C_VEL
LIN {X 0,Y 221.856,Z 401.875,A -85,B 0,C 180,E1 -20392.141,E2 -20392.141} C_VEL
LIN {X 0,Y 223.504,Z 404.074,A -85,B 0,C 180,E1 -20392.559,E2 -20392.559} C_VEL
LIN {X 0,Y 230.678,Z 416.044,A -85,B 0,C 180,E1 -20394.377,E2 -20394.377} C_VEL
LIN {X 0,Y 237.05,Z 428.891,A -85,B 0,C 180,E1 -20395.948,E2 -20395.948} C_VEL
LIN {X 0,Y 242.465,Z 441.813,A -85,B 0,C 180,E1 -20397.266,E2 -20397.266} C_VEL
LIN {X 0,Y 242.942,Z 443.202,A -85,B 0,C 180,E1 -20397.387,E2 -20397.387} C_VEL
LIN {X 0,Y 240.487,Z 503.645,A -85,B 0,C 180,E1 -20399.151,E2 -20399.151} C_VEL
LIN {X 0,Y 239.219,Z 517.421,A -85,B 0,C 180,E1 -20399.878,E2 -20399.878} C_VEL
LIN {X 0,Y 237.687,Z 530.177,A -85,B 0,C 180,E1 -20400.921,E2 -20400.921} C_VEL
LIN {X 0,Y 235.702,Z 541.968,A -85,B 0,C 180,E1 -20402.233,E2 -20402.233} C_VEL
LIN {X 0,Y 233.357,Z 553.295,A -85,B 0,C 180,E1 -20403.867,E2 -20403.867} C_VEL
LIN {X 0,Y 231.06,Z 563.345,A -85,B 0,C 180,E1 -20405.722,E2 -20405.722} C_VEL
LIN {X 0,Y 228.702,Z 572.646,A -85,B 0,C 180,E1 -20407.887,E2 -20407.887} C_VEL
LIN {X 0,Y 226.068,Z 581.543,A -85,B 0,C 180,E1 -20410.477,E2 -20410.477} C_VEL
LIN {X 0,Y 223.955,Z 588.696,A -85,B 0,C 180,E1 -20413.126,E2 -20413.126} C_VEL
LIN {X 0,Y 222.416,Z 593.52,A -85,B 0,C 180,E1 -20415.358,E2 -20415.358} C_VEL
LIN {X 0,Y 220.976,Z 598.203,A -85,B 0,C 180,E1 -20418.07,E2 -20418.07} C_VEL
LIN {X 0,Y 219.919,Z 601.785,A -85,B 0,C 180,E1 -20420.806,E2 -20420.806} C_VEL
LIN {X 0,Y 219.294,Z 604.287,A -85,B 0,C 180,E1 -20423.465,E2 -20423.465} C_VEL
LIN {X 0,Y 218.913,Z 606.005,A -85,B 0,C 180,E1 -20426.319,E2 -20426.319} C_VEL
LIN {X 0,Y 218.746,Z 606.839,A -85,B 0,C 180,E1 -20430,E2 -20430} C_VEL
LIN {X 0,Y 218.775,Z 606.646,A -85,B 0,C 180,E1 -20431.841,E2 -20431.841} C_VEL
LIN {X 0,Y 218.913,Z 606.061,A -85,B 0,C 180,E1 -20433.681,E2 -20433.681} C_VEL
LIN {X 0,Y 219.472,Z 603.744,A -85,B 0,C 180,E1 -20437.359,E2 -20437.359} C_VEL
LIN {X 0,Y 220.236,Z 600.884,A -85,B 0,C 180,E1 -20440.108,E2 -20440.108} C_VEL
LIN {X 0,Y 221.357,Z 597.002,A -85,B 0,C 180,E1 -20442.841,E2 -20442.841} C_VEL
LIN {X 0,Y 222.899,Z 591.991,A -85,B 0,C 180,E1 -20445.545,E2 -20445.545} C_VEL
LIN {X 0,Y 224.805,Z 585.677,A -85,B 0,C 180,E1 -20448.217,E2 -20448.217} C_VEL
LIN {X 0,Y 227.27,Z 577.768,A -85,B 0,C 180,E1 -20450.831,E2 -20450.831} C_VEL
LIN {X 0,Y 229.493,Z 569.782,A -85,B 0,C 180,E1 -20452.962,E2 -20452.962} C_VEL
LIN {X 0,Y 231.851,Z 559.873,A -85,B 0,C 180,E1 -20455.111,E2 -20455.111} C_VEL
LIN {X 0,Y 234.385,Z 548.787,A -85,B 0,C 180,E1 -20456.969,E2 -20456.969} C_VEL
LIN {X 0,Y 236.568,Z 537.913,A -85,B 0,C 180,E1 -20458.38,E2 -20458.38} C_VEL
LIN {X 0,Y 238.384,Z 525.897,A -85,B 0,C 180,E1 -20459.591,E2 -20459.591} C_VEL
LIN {X 0,Y 239.793,Z 514.031,A -85,B 0,C 180,E1 -20460.453,E2 -20460.453} C_VEL
LIN {X 0,Y 240.733,Z 501.257,A -85,B 0,C 180,E1 -20461.064,E2 -20461.064} C_VEL
LIN {X 0,Y 243.074,Z 443.311,A -85,B 0,C 180,E1 -20462.731,E2 -20462.731} C_VEL
LIN {X 0,Y 236.797,Z 428.207,A -85,B 0,C 180,E1 -20464.264,E2 -20464.264} C_VEL
LIN {X 0,Y 230.885,Z 416.381,A -85,B 0,C 180,E1 -20465.723,E2 -20465.723} C_VEL
LIN {X 0,Y 225.16,Z 406.81,A -85,B 0,C 180,E1 -20467.163,E2 -20467.163} C_VEL
LIN {X 0,Y 222.67,Z 402.934,A -85,B 0,C 180,E1 -20467.81,E2 -20467.81} C_VEL
LIN {X 0,Y 221.136,Z 400.316,A -85,B 0,C 180,E1 -20468.228,E2 -20468.228} C_VEL
LIN {X 0,Y 220.809,Z 398.979,A -85,B 0,C 180,E1 -20468.385,E2 -20468.385} C_VEL
LIN {X 0,Y 220.795,Z 398.978,A -85,B 0,C 180,E1 -20472.937,E2 -20472.937} C_VEL
LIN {X 0,Y 220.865,Z 398.951,A -85,B 0,C 180,E1 -20477.042,E2 -20477.042} C_VEL
LIN {X 0,Y 220.854,Z 398.974,A -85,B 0,C 180,E1 -20480.473,E2 -20480.473} C_VEL
LIN {X 0,Y 220.813,Z 398.98,A -85,B 0,C 180,E1 -20485.047,E2 -20485.047} C_VEL
LIN {X 0,Y 220.865,Z 398.974,A -85,B 0,C 180,E1 -20489.394,E2 -20489.394} C_VEL
LIN {X 0,Y 220.892,Z 398.97,A -85,B 0,C 180,E1 -20493.549,E2 -20493.549} C_VEL
LIN {X 0,Y 220.874,Z 398.964,A -85,B 0,C 180,E1 -20497.553,E2 -20497.553} C_VEL
LIN {X 0,Y 220.98,Z 398.946,A -85,B 0,C 180,E1 -20502.571,E2 -20502.571} C_VEL
LIN {X 0,Y 221.008,Z 398.951,A -85,B 0,C 180,E1 -20507.138,E2 -20507.138} C_VEL
LIN {X 0,Y 221.232,Z 398.923,A -85,B 0,C 180,E1 -20510.86,E2 -20510.86} C_VEL
LIN {X 0,Y 221.285,Z 398.921,A -85,B 0,C 180,E1 -20512.701,E2 -20512.701} C_VEL
LIN {X 0,Y 221.508,Z 398.892,A -85,B 0,C 180,E1 -20518.182,E2 -20518.182} C_VEL
LIN {X 0,Y 221.508,Z 398.878,A -85,B 0,C 180,E1 -20521.818,E2 -20521.818} C_VEL
LIN {X 0,Y 221.285,Z 398.911,A -85,B 0,C 180,E1 -20527.298,E2 -20527.298} C_VEL
LIN {X 0,Y 221.108,Z 398.942,A -85,B 0,C 180,E1 -20530.994,E2 -20530.994} C_VEL
LIN {X 0,Y 221.012,Z 398.953,A -85,B 0,C 180,E1 -20536.63,E2 -20536.63} C_VEL
LIN {X 0,Y 220.888,Z 398.961,A -85,B 0,C 180,E1 -20540.487,E2 -20540.487} C_VEL
LIN {X 0,Y 220.864,Z 398.966,A -85,B 0,C 180,E1 -20544.435,E2 -20544.435} C_VEL
LIN {X 0,Y 220.833,Z 398.976,A -85,B 0,C 180,E1 -20548.514,E2 -20548.514} C_VEL
LIN {X 0,Y 220.821,Z 398.97,A -85,B 0,C 180,E1 -20552.755,E2 -20552.755} C_VEL
LIN {X 0,Y 220.836,Z 398.967,A -85,B 0,C 180,E1 -20557.289,E2 -20557.289} C_VEL
LIN {X 0,Y 220.848,Z 398.968,A -85,B 0,C 180,E1 -20560.005,E2 -20560.005} C_VEL
LIN {X 0,Y 220.201,Z 399.076,A -85,B 0,C 180,E1 -20561.019,E2 -20561.019} C_VEL
LIN {X 0,Y 217.444,Z 399.395,A -85,B 0,C 180,E1 -20562.619,E2 -20562.619} C_VEL
LIN {X 0,Y 214.575,Z 399.752,A -85,B 0,C 180,E1 -20564.251,E2 -20564.251} C_VEL
LIN {X 0,Y 213.795,Z 399.873,A -85,B 0,C 180,E1 -20565.301,E2 -20565.301} C_VEL
LIN {X 0,Y 216,Z 408.337,A -85,B 0,C 180,E1 -20570.009,E2 -20570.009} C_VEL
LIN {X 0,Y 216.444,Z 409.836,A -85,B 0,C 180,E1 -20570.694,E2 -20570.694} C_VEL
LIN {X 0,Y 218.711,Z 414.124,A -85,B 0,C 180,E1 -20571.35,E2 -20571.35} C_VEL
LIN {X 0,Y 225.105,Z 426.982,A -85,B 0,C 180,E1 -20573.132,E2 -20573.132} C_VEL
LIN {X 0,Y 232.157,Z 443.064,A -85,B 0,C 180,E1 -20575.01,E2 -20575.01} C_VEL
LIN {X 0,Y 233.513,Z 446.948,A -85,B 0,C 180,E1 -20575.382,E2 -20575.382} C_VEL
LIN {X 0,Y 236.115,Z 466.566,A -85,B 0,C 180,E1 -20576.515,E2 -20576.515} C_VEL
LIN {X 0,Y 233.977,Z 519.419,A -85,B 0,C 180,E1 -20578.123,E2 -20578.123} C_VEL
LIN {X 0,Y 232.513,Z 533.069,A -85,B 0,C 180,E1 -20578.845,E2 -20578.845} C_VEL
LIN {X 0,Y 230.662,Z 545.284,A -85,B 0,C 180,E1 -20579.82,E2 -20579.82} C_VEL
LIN {X 0,Y 228.187,Z 557.962,A -85,B 0,C 180,E1 -20581.234,E2 -20581.234} C_VEL
LIN {X 0,Y 225.601,Z 569.243,A -85,B 0,C 180,E1 -20582.897,E2 -20582.897} C_VEL
LIN {X 0,Y 222.925,Z 579.407,A -85,B 0,C 180,E1 -20584.812,E2 -20584.812} C_VEL
LIN {X 0,Y 220.254,Z 588.567,A -85,B 0,C 180,E1 -20586.991,E2 -20586.991} C_VEL
LIN {X 0,Y 218.147,Z 596.149,A -85,B 0,C 180,E1 -20589.245,E2 -20589.245} C_VEL
LIN {X 0,Y 215.911,Z 603.59,A -85,B 0,C 180,E1 -20591.988,E2 -20591.988} C_VEL
LIN {X 0,Y 214.111,Z 609.57,A -85,B 0,C 180,E1 -20594.776,E2 -20594.776} C_VEL
LIN {X 0,Y 212.811,Z 614.301,A -85,B 0,C 180,E1 -20597.605,E2 -20597.605} C_VEL
LIN {X 0,Y 212.031,Z 617.924,A -85,B 0,C 180,E1 -20600.461,E2 -20600.461} C_VEL
LIN {X 0,Y 211.68,Z 619.792,A -85,B 0,C 180,E1 -20602.369,E2 -20602.369} C_VEL
LIN {X 0,Y 211.42,Z 622.016,A -85,B 0,C 180,E1 -20605.759,E2 -20605.759} C_VEL
LIN {X 0,Y 211.514,Z 622.817,A -85,B 0,C 180,E1 -20608.096,E2 -20608.096} C_VEL
LIN {X 0,Y 211.64,Z 623.035,A -85,B 0,C 180,E1 -20610,E2 -20610} C_VEL
LIN {X 0,Y 211.516,Z 622.806,A -85,B 0,C 180,E1 -20611.904,E2 -20611.904} C_VEL
LIN {X 0,Y 211.473,Z 621.917,A -85,B 0,C 180,E1 -20614.434,E2 -20614.434} C_VEL
LIN {X 0,Y 211.659,Z 619.755,A -85,B 0,C 180,E1 -20617.632,E2 -20617.632} C_VEL
LIN {X 0,Y 212.239,Z 616.792,A -85,B 0,C 180,E1 -20620.493,E2 -20620.493} C_VEL
LIN {X 0,Y 213.143,Z 612.786,A -85,B 0,C 180,E1 -20623.345,E2 -20623.345} C_VEL
LIN {X 0,Y 215.002,Z 606.646,A -85,B 0,C 180,E1 -20626.619,E2 -20626.619} C_VEL
LIN {X 0,Y 217.067,Z 599.946,A -85,B 0,C 180,E1 -20629.382,E2 -20629.382} C_VEL
LIN {X 0,Y 219.408,Z 591.629,A -85,B 0,C 180,E1 -20632.11,E2 -20632.11} C_VEL
LIN {X 0,Y 221.802,Z 583.115,A -85,B 0,C 180,E1 -20634.325,E2 -20634.325} C_VEL
LIN {X 0,Y 224.69,Z 572.603,A -85,B 0,C 180,E1 -20636.469,E2 -20636.469} C_VEL
LIN {X 0,Y 227.525,Z 560.771,A -85,B 0,C 180,E1 -20638.353,E2 -20638.353} C_VEL
LIN {X 0,Y 229.929,Z 548.851,A -85,B 0,C 180,E1 -20639.781,E2 -20639.781} C_VEL
LIN {X 0,Y 231.942,Z 536.446,A -85,B 0,C 180,E1 -20640.878,E2 -20640.878} C_VEL
LIN {X 0,Y 233.437,Z 524.008,A -85,B 0,C 180,E1 -20641.643,E2 -20641.643} C_VEL
LIN {X 0,Y 234.342,Z 510.753,A -85,B 0,C 180,E1 -20642.139,E2 -20642.139} C_VEL
LIN {X 0,Y 236.019,Z 466.644,A -85,B 0,C 180,E1 -20643.443,E2 -20643.443} C_VEL
LIN {X 0,Y 233.21,Z 445.823,A -85,B 0,C 180,E1 -20644.652,E2 -20644.652} C_VEL
LIN {X 0,Y 227.769,Z 432.902,A -85,B 0,C 180,E1 -20646.084,E2 -20646.084} C_VEL
LIN {X 0,Y 220.865,Z 418.285,A -85,B 0,C 180,E1 -20647.973,E2 -20647.973} C_VEL
LIN {X 0,Y 216.459,Z 409.847,A -85,B 0,C 180,E1 -20649.231,E2 -20649.231} C_VEL
LIN {X 0,Y 214.745,Z 403.443,A -85,B 0,C 180,E1 -20652.579,E2 -20652.579} C_VEL
LIN {X 0,Y 213.781,Z 399.834,A -85,B 0,C 180,E1 -20654.691,E2 -20654.691} C_VEL
LIN {X 0,Y 213.793,Z 399.848,A -85,B 0,C 180,E1 -20659.118,E2 -20659.118} C_VEL
LIN {X 0,Y 213.752,Z 399.856,A -85,B 0,C 180,E1 -20663.713,E2 -20663.713} C_VEL
LIN {X 0,Y 213.793,Z 399.852,A -85,B 0,C 180,E1 -20668.724,E2 -20668.724} C_VEL
LIN {X 0,Y 213.823,Z 399.843,A -85,B 0,C 180,E1 -20672.603,E2 -20672.603} C_VEL
LIN {X 0,Y 213.848,Z 399.832,A -85,B 0,C 180,E1 -20676.953,E2 -20676.953} C_VEL
LIN {X 0,Y 213.939,Z 399.82,A -85,B 0,C 180,E1 -20682.803,E2 -20682.803} C_VEL
LIN {X 0,Y 213.949,Z 399.835,A -85,B 0,C 180,E1 -20686.706,E2 -20686.706} C_VEL
LIN {X 0,Y 214.163,Z 399.793,A -85,B 0,C 180,E1 -20690.556,E2 -20690.556} C_VEL
LIN {X 0,Y 214.223,Z 399.798,A -85,B 0,C 180,E1 -20692.46,E2 -20692.46} C_VEL
LIN {X 0,Y 214.441,Z 399.759,A -85,B 0,C 180,E1 -20698.122,E2 -20698.122} C_VEL
LIN {X 0,Y 214.55,Z 399.758,A -85,B 0,C 180,E1 -20700,E2 -20700} C_VEL
LIN {X 0,Y 214.441,Z 399.771,A -85,B 0,C 180,E1 -20701.878,E2 -20701.878} C_VEL
LIN {X 0,Y 214.236,Z 399.798,A -85,B 0,C 180,E1 -20707.54,E2 -20707.54} C_VEL
LIN {X 0,Y 214.019,Z 399.812,A -85,B 0,C 180,E1 -20711.363,E2 -20711.363} C_VEL
LIN {X 0,Y 213.929,Z 399.837,A -85,B 0,C 180,E1 -20715.237,E2 -20715.237} C_VEL
LIN {X 0,Y 213.835,Z 399.832,A -85,B 0,C 180,E1 -20719.188,E2 -20719.188} C_VEL
LIN {X 0,Y 213.844,Z 399.847,A -85,B 0,C 180,E1 -20723.228,E2 -20723.228} C_VEL
LIN {X 0,Y 213.826,Z 399.845,A -85,B 0,C 180,E1 -20727.45,E2 -20727.45} C_VEL
LIN {X 0,Y 213.777,Z 399.844,A -85,B 0,C 180,E1 -20731.736,E2 -20731.736} C_VEL
LIN {X 0,Y 213.752,Z 399.851,A -85,B 0,C 180,E1 -20736.287,E2 -20736.287} C_VEL
LIN {X 0,Y 213.792,Z 399.846,A -85,B 0,C 180,E1 -20741.107,E2 -20741.107} C_VEL
LIN {X 0,Y 213.807,Z 399.851,A -85,B 0,C 180,E1 -20743.686,E2 -20743.686} C_VEL
LIN {X 0,Y 213.747,Z 399.86,A -85,B 0,C 180,E1 -20746.333,E2 -20746.333} C_VEL
LIN {X 0,Y 213.778,Z 399.967,A -85,B 0,C 180,E1 -20750.338,E2 -20750.338} C_VEL
LIN {X 0,Y 214.854,Z 402.849,A -85,B 0,C 180,E1 -20750.7,E2 -20750.7} C_VEL
LIN {X 0,Y 216.552,Z 404.988,A -85,B 0,C 180,E1 -20751.16,E2 -20751.16} C_VEL
LIN {X 0,Y 218.642,Z 408.294,A -85,B 0,C 180,E1 -20751.741,E2 -20751.741} C_VEL
LIN {X 0,Y 226.688,Z 421.829,A -85,B 0,C 180,E1 -20753.867,E2 -20753.867} C_VEL
LIN {X 0,Y 233.95,Z 437.389,A -85,B 0,C 180,E1 -20755.739,E2 -20755.739} C_VEL
LIN {X 0,Y 236.932,Z 444.984,A -85,B 0,C 180,E1 -20756.505,E2 -20756.505} C_VEL
LIN {X 0,Y 234.452,Z 503.642,A -85,B 0,C 180,E1 -20758.25,E2 -20758.25} C_VEL
LIN {X 0,Y 233.209,Z 517.121,A -85,B 0,C 180,E1 -20758.97,E2 -20758.97} C_VEL
LIN {X 0,Y 231.711,Z 529.365,A -85,B 0,C 180,E1 -20759.97,E2 -20759.97} C_VEL
LIN {X 0,Y 229.786,Z 540.658,A -85,B 0,C 180,E1 -20761.203,E2 -20761.203} C_VEL
LIN {X 0,Y 227.3,Z 552.28,A -85,B 0,C 180,E1 -20762.867,E2 -20762.867} C_VEL
LIN {X 0,Y 224.764,Z 563.03,A -85,B 0,C 180,E1 -20764.859,E2 -20764.859} C_VEL
LIN {X 0,Y 222.147,Z 572.916,A -85,B 0,C 180,E1 -20767.198,E2 -20767.198} C_VEL
LIN {X 0,Y 219.4,Z 581.812,A -85,B 0,C 180,E1 -20769.858,E2 -20769.858} C_VEL
LIN {X 0,Y 217.147,Z 588.966,A -85,B 0,C 180,E1 -20772.58,E2 -20772.58} C_VEL
LIN {X 0,Y 215.538,Z 593.789,A -85,B 0,C 180,E1 -20774.88,E2 -20774.88} C_VEL
LIN {X 0,Y 214.025,Z 598.472,A -85,B 0,C 180,E1 -20777.676,E2 -20777.676} C_VEL
LIN {X 0,Y 212.907,Z 602.053,A -85,B 0,C 180,E1 -20780.5,E2 -20780.5} C_VEL
LIN {X 0,Y 212.181,Z 604.79,A -85,B 0,C 180,E1 -20783.559,E2 -20783.559} C_VEL
LIN {X 0,Y 211.845,Z 606.271,A -85,B 0,C 180,E1 -20786.196,E2 -20786.196} C_VEL
LIN {X 0,Y 211.66,Z 607.106,A -85,B 0,C 180,E1 -20790,E2 -20790} C_VEL
LIN {X 0,Y 211.694,Z 606.912,A -85,B 0,C 180,E1 -20791.902,E2 -20791.902} C_VEL
LIN {X 0,Y 211.844,Z 606.327,A -85,B 0,C 180,E1 -20793.804,E2 -20793.804} C_VEL
LIN {X 0,Y 212.448,Z 604.01,A -85,B 0,C 180,E1 -20797.604,E2 -20797.604} C_VEL
LIN {X 0,Y 213.252,Z 601.15,A -85,B 0,C 180,E1 -20800.443,E2 -20800.443} C_VEL
LIN {X 0,Y 214.442,Z 597.268,A -85,B 0,C 180,E1 -20803.262,E2 -20803.262} C_VEL
LIN {X 0,Y 216.068,Z 592.256,A -85,B 0,C 180,E1 -20806.05,E2 -20806.05} C_VEL
LIN {X 0,Y 218.07,Z 585.942,A -85,B 0,C 180,E1 -20808.801,E2 -20808.801} C_VEL
LIN {X 0,Y 220.662,Z 578.032,A -85,B 0,C 180,E1 -20811.485,E2 -20811.485} C_VEL
LIN {X 0,Y 223.102,Z 569.543,A -85,B 0,C 180,E1 -20813.799,E2 -20813.799} C_VEL
LIN {X 0,Y 225.448,Z 560.137,A -85,B 0,C 180,E1 -20815.876,E2 -20815.876} C_VEL
LIN {X 0,Y 227.786,Z 550.443,A -85,B 0,C 180,E1 -20817.567,E2 -20817.567} C_VEL
LIN {X 0,Y 230.032,Z 539.935,A -85,B 0,C 180,E1 -20819.013,E2 -20819.013} C_VEL
LIN {X 0,Y 232.102,Z 527.283,A -85,B 0,C 180,E1 -20820.35,E2 -20820.35} C_VEL
LIN {X 0,Y 233.684,Z 514.537,A -85,B 0,C 180,E1 -20821.318,E2 -20821.318} C_VEL
LIN {X 0,Y 234.708,Z 501.241,A -85,B 0,C 180,E1 -20821.965,E2 -20821.965} C_VEL
LIN {X 0,Y 237.037,Z 445.078,A -85,B 0,C 180,E1 -20823.619,E2 -20823.619} C_VEL
LIN {X 0,Y 231.029,Z 430.712,A -85,B 0,C 180,E1 -20825.16,E2 -20825.16} C_VEL
LIN {X 0,Y 225.329,Z 419.354,A -85,B 0,C 180,E1 -20826.639,E2 -20826.639} C_VEL
LIN {X 0,Y 218.298,Z 407.886,A -85,B 0,C 180,E1 -20828.509,E2 -20828.509} C_VEL
LIN {X 0,Y 215.901,Z 404.113,A -85,B 0,C 180,E1 -20829.18,E2 -20829.18} C_VEL
LIN {X 0,Y 214.19,Z 401.557,A -85,B 0,C 180,E1 -20829.667,E2 -20829.667} C_VEL
LIN {X 0,Y 213.764,Z 399.856,A -85,B 0,C 180,E1 -20829.852,E2 -20829.852} C_VEL
LIN {X 0,Y 213.747,Z 399.859,A -85,B 0,C 180,E1 -20833.667,E2 -20833.667} C_VEL
LIN {X 0,Y 213.781,Z 399.835,A -85,B 0,C 180,E1 -20836.34,E2 -20836.34} C_VEL
LIN {X 0,Y 213.793,Z 399.845,A -85,B 0,C 180,E1 -20839.118,E2 -20839.118} C_VEL
LIN {X 0,Y 213.752,Z 399.856,A -85,B 0,C 180,E1 -20843.713,E2 -20843.713} C_VEL
LIN {X 0,Y 213.793,Z 399.853,A -85,B 0,C 180,E1 -20848.724,E2 -20848.724} C_VEL
LIN {X 0,Y 213.823,Z 399.846,A -85,B 0,C 180,E1 -20852.603,E2 -20852.603} C_VEL
LIN {X 0,Y 213.849,Z 399.836,A -85,B 0,C 180,E1 -20856.952,E2 -20856.952} C_VEL
LIN {X 0,Y 213.94,Z 399.823,A -85,B 0,C 180,E1 -20862.803,E2 -20862.803} C_VEL
LIN {X 0,Y 213.949,Z 399.834,A -85,B 0,C 180,E1 -20866.706,E2 -20866.706} C_VEL
LIN {X 0,Y 214.163,Z 399.802,A -85,B 0,C 180,E1 -20870.556,E2 -20870.556} C_VEL
LIN {X 0,Y 214.223,Z 399.8,A -85,B 0,C 180,E1 -20872.459,E2 -20872.459} C_VEL
LIN {X 0,Y 214.441,Z 399.772,A -85,B 0,C 180,E1 -20878.122,E2 -20878.122} C_VEL
LIN {X 0,Y 214.55,Z 399.757,A -85,B 0,C 180,E1 -20880,E2 -20880} C_VEL
LIN {X 0,Y 214.442,Z 399.757,A -85,B 0,C 180,E1 -20881.878,E2 -20881.878} C_VEL
LIN {X 0,Y 214.223,Z 399.789,A -85,B 0,C 180,E1 -20887.54,E2 -20887.54} C_VEL
LIN {X 0,Y 214.041,Z 399.822,A -85,B 0,C 180,E1 -20891.362,E2 -20891.362} C_VEL
LIN {X 0,Y 213.929,Z 399.828,A -85,B 0,C 180,E1 -20895.237,E2 -20895.237} C_VEL
LIN {X 0,Y 213.835,Z 399.839,A -85,B 0,C 180,E1 -20899.188,E2 -20899.188} C_VEL
LIN {X 0,Y 213.844,Z 399.845,A -85,B 0,C 180,E1 -20903.227,E2 -20903.227} C_VEL
LIN {X 0,Y 213.826,Z 399.849,A -85,B 0,C 180,E1 -20907.45,E2 -20907.45} C_VEL
LIN {X 0,Y 213.776,Z 399.853,A -85,B 0,C 180,E1 -20911.736,E2 -20911.736} C_VEL
LIN {X 0,Y 213.752,Z 399.852,A -85,B 0,C 180,E1 -20916.287,E2 -20916.287} C_VEL
LIN {X 0,Y 213.792,Z 399.847,A -85,B 0,C 180,E1 -20921.107,E2 -20921.107} C_VEL
LIN {X 0,Y 213.795,Z 399.873,A -85,B 0,C 180,E1 -20925.301,E2 -20925.301} C_VEL
LIN {X 0,Y 213.125,Z 402.205,A -85,B 0,C 180,E1 -20926.341,E2 -20926.341} C_VEL
LIN {X 0,Y 210.66,Z 406.878,A -85,B 0,C 180,E1 -20928.033,E2 -20928.033} C_VEL
LIN {X 0,Y 210.096,Z 410.657,A -85,B 0,C 180,E1 -20929.02,E2 -20929.02} C_VEL
LIN {X 0,Y 211.009,Z 413.201,A -85,B 0,C 180,E1 -20929.63,E2 -20929.63} C_VEL
LIN {X 0,Y 211.167,Z 413.416,A -85,B 0,C 180,E1 -20929.678,E2 -20929.678} C_VEL
LIN {X 0,Y 216.781,Z 423.988,A -85,B 0,C 180,E1 -20931.354,E2 -20931.354} C_VEL
LIN {X 0,Y 223.913,Z 439.426,A -85,B 0,C 180,E1 -20933.392,E2 -20933.392} C_VEL
LIN {X 0,Y 227.781,Z 449.012,A -85,B 0,C 180,E1 -20934.468,E2 -20934.468} C_VEL
LIN {X 0,Y 230.21,Z 468.061,A -85,B 0,C 180,E1 -20935.602,E2 -20935.602} C_VEL
LIN {X 0,Y 228.044,Z 518.67,A -85,B 0,C 180,E1 -20937.163,E2 -20937.163} C_VEL
LIN {X 0,Y 226.571,Z 532.192,A -85,B 0,C 180,E1 -20937.879,E2 -20937.879} C_VEL
LIN {X 0,Y 224.531,Z 545.022,A -85,B 0,C 180,E1 -20938.905,E2 -20938.905} C_VEL
LIN {X 0,Y 221.99,Z 557.7,A -85,B 0,C 180,E1 -20940.353,E2 -20940.353} C_VEL
LIN {X 0,Y 219.279,Z 568.978,A -85,B 0,C 180,E1 -20942.048,E2 -20942.048} C_VEL
LIN {X 0,Y 216.504,Z 579.142,A -85,B 0,C 180,E1 -20944.01,E2 -20944.01} C_VEL
LIN {X 0,Y 213.72,Z 588.302,A -85,B 0,C 180,E1 -20946.245,E2 -20946.245} C_VEL
LIN {X 0,Y 211.186,Z 596.916,A -85,B 0,C 180,E1 -20948.915,E2 -20948.915} C_VEL
LIN {X 0,Y 208.826,Z 604.442,A -85,B 0,C 180,E1 -20951.862,E2 -20951.862} C_VEL
LIN {X 0,Y 206.69,Z 610.999,A -85,B 0,C 180,E1 -20955.226,E2 -20955.226} C_VEL
LIN {X 0,Y 205.503,Z 615.348,A -85,B 0,C 180,E1 -20958.159,E2 -20958.159} C_VEL
LIN {X 0,Y 204.987,Z 617.655,A -85,B 0,C 180,E1 -20960.13,E2 -20960.13} C_VEL
LIN {X 0,Y 204.631,Z 619.525,A -85,B 0,C 180,E1 -20962.104,E2 -20962.104} C_VEL
LIN {X 0,Y 204.352,Z 621.842,A -85,B 0,C 180,E1 -20965.834,E2 -20965.834} C_VEL
LIN {X 0,Y 204.412,Z 622.55,A -85,B 0,C 180,E1 -20968.03,E2 -20968.03} C_VEL
LIN {X 0,Y 204.554,Z 622.769,A -85,B 0,C 180,E1 -20970,E2 -20970} C_VEL
LIN {X 0,Y 204.414,Z 622.538,A -85,B 0,C 180,E1 -20971.97,E2 -20971.97} C_VEL
LIN {X 0,Y 204.384,Z 621.774,A -85,B 0,C 180,E1 -20974.287,E2 -20974.287} C_VEL
LIN {X 0,Y 204.615,Z 619.487,A -85,B 0,C 180,E1 -20977.897,E2 -20977.897} C_VEL
LIN {X 0,Y 205.214,Z 616.522,A -85,B 0,C 180,E1 -20980.857,E2 -20980.857} C_VEL
LIN {X 0,Y 206.2,Z 612.516,A -85,B 0,C 180,E1 -20983.803,E2 -20983.803} C_VEL
LIN {X 0,Y 208.194,Z 606.377,A -85,B 0,C 180,E1 -20987.179,E2 -20987.179} C_VEL
LIN {X 0,Y 210.35,Z 599.676,A -85,B 0,C 180,E1 -20990.026,E2 -20990.026} C_VEL
LIN {X 0,Y 212.755,Z 591.511,A -85,B 0,C 180,E1 -20992.787,E2 -20992.787} C_VEL
LIN {X 0,Y 215.344,Z 582.845,A -85,B 0,C 180,E1 -20995.104,E2 -20995.104} C_VEL
LIN {X 0,Y 218.345,Z 572.332,A -85,B 0,C 180,E1 -20997.301,E2 -20997.301} C_VEL
LIN {X 0,Y 221.299,Z 560.5,A -85,B 0,C 180,E1 -20999.227,E2 -20999.227} C_VEL
LIN {X 0,Y 223.793,Z 548.578,A -85,B 0,C 180,E1 -21000.684,E2 -21000.684} C_VEL
LIN {X 0,Y 225.882,Z 536.171,A -85,B 0,C 180,E1 -21001.801,E2 -21001.801} C_VEL
LIN {X 0,Y 227.482,Z 523.21,A -85,B 0,C 180,E1 -21002.607,E2 -21002.607} C_VEL
LIN {X 0,Y 228.459,Z 508.392,A -85,B 0,C 180,E1 -21003.147,E2 -21003.147} C_VEL
LIN {X 0,Y 230.072,Z 467.563,A -85,B 0,C 180,E1 -21004.382,E2 -21004.382} C_VEL
LIN {X 0,Y 227.516,Z 448.337,A -85,B 0,C 180,E1 -21005.544,E2 -21005.544} C_VEL
LIN {X 0,Y 221.691,Z 434.422,A -85,B 0,C 180,E1 -21007.165,E2 -21007.165} C_VEL
LIN {X 0,Y 215.481,Z 421.514,A -85,B 0,C 180,E1 -21008.952,E2 -21008.952} C_VEL
LIN {X 0,Y 210.783,Z 412.772,A -85,B 0,C 180,E1 -21010.361,E2 -21010.361} C_VEL
LIN {X 0,Y 208.967,Z 409.085,A -85,B 0,C 180,E1 -21011.008,E2 -21011.008} C_VEL
LIN {X 0,Y 207.312,Z 402.865,A -85,B 0,C 180,E1 -21014.609,E2 -21014.609} C_VEL
LIN {X 0,Y 206.773,Z 400.706,A -85,B 0,C 180,E1 -21016.027,E2 -21016.027} C_VEL
LIN {X 0,Y 206.758,Z 400.73,A -85,B 0,C 180,E1 -21021.424,E2 -21021.424} C_VEL
LIN {X 0,Y 206.729,Z 400.734,A -85,B 0,C 180,E1 -21024.694,E2 -21024.694} C_VEL
LIN {X 0,Y 206.721,Z 400.733,A -85,B 0,C 180,E1 -21029.339,E2 -21029.339} C_VEL
LIN {X 0,Y 206.73,Z 400.732,A -85,B 0,C 180,E1 -21033.772,E2 -21033.772} C_VEL
LIN {X 0,Y 206.754,Z 400.721,A -85,B 0,C 180,E1 -21038.043,E2 -21038.043} C_VEL
LIN {X 0,Y 206.869,Z 400.702,A -85,B 0,C 180,E1 -21042.196,E2 -21042.196} C_VEL
LIN {X 0,Y 206.891,Z 400.713,A -85,B 0,C 180,E1 -21046.244,E2 -21046.244} C_VEL
LIN {X 0,Y 207.101,Z 400.67,A -85,B 0,C 180,E1 -21050.231,E2 -21050.231} C_VEL
LIN {X 0,Y 207.163,Z 400.677,A -85,B 0,C 180,E1 -21052.201,E2 -21052.201} C_VEL
LIN {X 0,Y 207.378,Z 400.638,A -85,B 0,C 180,E1 -21058.058,E2 -21058.058} C_VEL
LIN {X 0,Y 207.514,Z 400.634,A -85,B 0,C 180,E1 -21060,E2 -21060} C_VEL
LIN {X 0,Y 207.081,Z 400.674,A -85,B 0,C 180,E1 -21063.892,E2 -21063.892} C_VEL
LIN {X 0,Y 207.174,Z 400.677,A -85,B 0,C 180,E1 -21067.799,E2 -21067.799} C_VEL
LIN {X 0,Y 206.939,Z 400.69,A -85,B 0,C 180,E1 -21071.758,E2 -21071.758} C_VEL
LIN {X 0,Y 206.862,Z 400.717,A -85,B 0,C 180,E1 -21075.771,E2 -21075.771} C_VEL
LIN {X 0,Y 206.78,Z 400.711,A -85,B 0,C 180,E1 -21079.87,E2 -21079.87} C_VEL
LIN {X 0,Y 206.76,Z 400.726,A -85,B 0,C 180,E1 -21084.073,E2 -21084.073} C_VEL
LIN {X 0,Y 206.741,Z 400.732,A -85,B 0,C 180,E1 -21088.419,E2 -21088.419} C_VEL
LIN {X 0,Y 206.707,Z 400.73,A -85,B 0,C 180,E1 -21092.956,E2 -21092.956} C_VEL
LIN {X 0,Y 206.723,Z 400.729,A -85,B 0,C 180,E1 -21097.731,E2 -21097.731} C_VEL
LIN {X 0,Y 206.722,Z 400.728,A -85,B 0,C 180,E1 -21101.589,E2 -21101.589} C_VEL
LIN {X 0,Y 206.673,Z 400.736,A -85,B 0,C 180,E1 -21105.571,E2 -21105.571} C_VEL
LIN {X 0,Y 206.697,Z 400.839,A -85,B 0,C 180,E1 -21108.713,E2 -21108.713} C_VEL
LIN {X 0,Y 207.655,Z 403.543,A -85,B 0,C 180,E1 -21109.069,E2 -21109.069} C_VEL
LIN {X 0,Y 209.597,Z 405.968,A -85,B 0,C 180,E1 -21109.639,E2 -21109.639} C_VEL
LIN {X 0,Y 211.858,Z 409.408,A -85,B 0,C 180,E1 -21110.312,E2 -21110.312} C_VEL
LIN {X 0,Y 220.138,Z 423.023,A -85,B 0,C 180,E1 -21112.647,E2 -21112.647} C_VEL
LIN {X 0,Y 225.221,Z 433.139,A -85,B 0,C 180,E1 -21114.031,E2 -21114.031} C_VEL
LIN {X 0,Y 230.742,Z 446.182,A -85,B 0,C 180,E1 -21115.515,E2 -21115.515} C_VEL
LIN {X 0,Y 231.095,Z 447.779,A -85,B 0,C 180,E1 -21115.635,E2 -21115.635} C_VEL
LIN {X 0,Y 228.485,Z 503.763,A -85,B 0,C 180,E1 -21117.31,E2 -21117.31} C_VEL
LIN {X 0,Y 227.167,Z 517.495,A -85,B 0,C 180,E1 -21118.057,E2 -21118.057} C_VEL
LIN {X 0,Y 225.607,Z 529.639,A -85,B 0,C 180,E1 -21119.07,E2 -21119.07} C_VEL
LIN {X 0,Y 223.614,Z 540.93,A -85,B 0,C 180,E1 -21120.33,E2 -21120.33} C_VEL
LIN {X 0,Y 221.006,Z 552.552,A -85,B 0,C 180,E1 -21122.028,E2 -21122.028} C_VEL
LIN {X 0,Y 218.342,Z 563.301,A -85,B 0,C 180,E1 -21124.065,E2 -21124.065} C_VEL
LIN {X 0,Y 215.614,Z 573.234,A -85,B 0,C 180,E1 -21126.482,E2 -21126.482} C_VEL
LIN {X 0,Y 212.762,Z 582.08,A -85,B 0,C 180,E1 -21129.201,E2 -21129.201} C_VEL
LIN {X 0,Y 210.375,Z 589.235,A -85,B 0,C 180,E1 -21132.001,E2 -21132.001} C_VEL
LIN {X 0,Y 208.68,Z 594.058,A -85,B 0,C 180,E1 -21134.37,E2 -21134.37} C_VEL
LIN {X 0,Y 207.096,Z 598.74,A -85,B 0,C 180,E1 -21137.257,E2 -21137.257} C_VEL
LIN {X 0,Y 205.92,Z 602.32,A -85,B 0,C 180,E1 -21140.175,E2 -21140.175} C_VEL
LIN {X 0,Y 205.069,Z 605.289,A -85,B 0,C 180,E1 -21143.655,E2 -21143.655} C_VEL
LIN {X 0,Y 204.76,Z 606.539,A -85,B 0,C 180,E1 -21146.064,E2 -21146.064} C_VEL
LIN {X 0,Y 204.616,Z 607.145,A -85,B 0,C 180,E1 -21148.032,E2 -21148.032} C_VEL
LIN {X 0,Y 204.577,Z 607.372,A -85,B 0,C 180,E1 -21150,E2 -21150} C_VEL
LIN {X 0,Y 204.615,Z 607.179,A -85,B 0,C 180,E1 -21151.968,E2 -21151.968} C_VEL
LIN {X 0,Y 205.029,Z 605.629,A -85,B 0,C 180,E1 -21155.902,E2 -21155.902} C_VEL
LIN {X 0,Y 205.416,Z 604.276,A -85,B 0,C 180,E1 -21157.866,E2 -21157.866} C_VEL
LIN {X 0,Y 206.268,Z 601.416,A -85,B 0,C 180,E1 -21160.801,E2 -21160.801} C_VEL
LIN {X 0,Y 207.544,Z 597.534,A -85,B 0,C 180,E1 -21163.711,E2 -21163.711} C_VEL
LIN {X 0,Y 209.259,Z 592.522,A -85,B 0,C 180,E1 -21166.587,E2 -21166.587} C_VEL
LIN {X 0,Y 211.361,Z 586.208,A -85,B 0,C 180,E1 -21169.421,E2 -21169.421} C_VEL
LIN {X 0,Y 214.084,Z 578.296,A -85,B 0,C 180,E1 -21172.18,E2 -21172.18} C_VEL
LIN {X 0,Y 216.479,Z 570.319,A -85,B 0,C 180,E1 -21174.427,E2 -21174.427} C_VEL
LIN {X 0,Y 219.09,Z 560.4,A -85,B 0,C 180,E1 -21176.685,E2 -21176.685} C_VEL
LIN {X 0,Y 221.522,Z 550.706,A -85,B 0,C 180,E1 -21178.416,E2 -21178.416} C_VEL
LIN {X 0,Y 223.867,Z 540.195,A -85,B 0,C 180,E1 -21179.892,E2 -21179.892} C_VEL
LIN {X 0,Y 226.025,Z 527.541,A -85,B 0,C 180,E1 -21181.256,E2 -21181.256} C_VEL
LIN {X 0,Y 227.617,Z 515.038,A -85,B 0,C 180,E1 -21182.231,E2 -21182.231} C_VEL
LIN {X 0,Y 228.67,Z 502.643,A -85,B 0,C 180,E1 -21182.864,E2 -21182.864} C_VEL
LIN {X 0,Y 231.098,Z 446.926,A -85,B 0,C 180,E1 -21184.545,E2 -21184.545} C_VEL
LIN {X 0,Y 225.25,Z 433.153,A -85,B 0,C 180,E1 -21186.117,E2 -21186.117} C_VEL
LIN {X 0,Y 220.272,Z 423.148,A -85,B 0,C 180,E1 -21187.479,E2 -21187.479} C_VEL
LIN {X 0,Y 213.591,Z 412.266,A -85,B 0,C 180,E1 -21189.342,E2 -21189.342} C_VEL
LIN {X 0,Y 209.484,Z 405.682,A -85,B 0,C 180,E1 -21190.569,E2 -21190.569} C_VEL
LIN {X 0,Y 207.352,Z 402.994,A -85,B 0,C 180,E1 -21191.201,E2 -21191.201} C_VEL
LIN {X 0,Y 206.672,Z 400.743,A -85,B 0,C 180,E1 -21191.498,E2 -21191.498} C_VEL
LIN {X 0,Y 206.707,Z 400.723,A -85,B 0,C 180,E1 -21195.56,E2 -21195.56} C_VEL
LIN {X 0,Y 206.723,Z 400.731,A -85,B 0,C 180,E1 -21199.763,E2 -21199.763} C_VEL
LIN {X 0,Y 206.723,Z 400.727,A -85,B 0,C 180,E1 -21202.269,E2 -21202.269} C_VEL
LIN {X 0,Y 206.707,Z 400.728,A -85,B 0,C 180,E1 -21207.044,E2 -21207.044} C_VEL
LIN {X 0,Y 206.764,Z 400.722,A -85,B 0,C 180,E1 -21212.096,E2 -21212.096} C_VEL
LIN {X 0,Y 206.782,Z 400.716,A -85,B 0,C 180,E1 -21216.583,E2 -21216.583} C_VEL
LIN {X 0,Y 206.87,Z 400.704,A -85,B 0,C 180,E1 -21222.196,E2 -21222.196} C_VEL
LIN {X 0,Y 206.891,Z 400.713,A -85,B 0,C 180,E1 -21226.244,E2 -21226.244} C_VEL
LIN {X 0,Y 207.102,Z 400.681,A -85,B 0,C 180,E1 -21230.231,E2 -21230.231} C_VEL
LIN {X 0,Y 207.164,Z 400.679,A -85,B 0,C 180,E1 -21232.201,E2 -21232.201} C_VEL
LIN {X 0,Y 207.378,Z 400.652,A -85,B 0,C 180,E1 -21238.058,E2 -21238.058} C_VEL
LIN {X 0,Y 207.514,Z 400.633,A -85,B 0,C 180,E1 -21240,E2 -21240} C_VEL
LIN {X 0,Y 207.379,Z 400.637,A -85,B 0,C 180,E1 -21241.942,E2 -21241.942} C_VEL
LIN {X 0,Y 207.164,Z 400.667,A -85,B 0,C 180,E1 -21247.799,E2 -21247.799} C_VEL
LIN {X 0,Y 206.978,Z 400.701,A -85,B 0,C 180,E1 -21251.755,E2 -21251.755} C_VEL
LIN {X 0,Y 206.863,Z 400.713,A -85,B 0,C 180,E1 -21255.771,E2 -21255.771} C_VEL
LIN {X 0,Y 206.78,Z 400.716,A -85,B 0,C 180,E1 -21259.869,E2 -21259.869} C_VEL
LIN {X 0,Y 206.76,Z 400.723,A -85,B 0,C 180,E1 -21264.073,E2 -21264.073} C_VEL
LIN {X 0,Y 206.741,Z 400.731,A -85,B 0,C 180,E1 -21268.419,E2 -21268.419} C_VEL
LIN {X 0,Y 206.706,Z 400.726,A -85,B 0,C 180,E1 -21272.956,E2 -21272.956} C_VEL
LIN {X 0,Y 206.723,Z 400.725,A -85,B 0,C 180,E1 -21277.731,E2 -21277.731} C_VEL
LIN {X 0,Y 206.722,Z 400.731,A -85,B 0,C 180,E1 -21281.589,E2 -21281.589} C_VEL
LIN {X 0,Y 206.788,Z 400.933,A -85,B 0,C 180,E1 -21284.127,E2 -21284.127} C_VEL
LIN {X 0,Y 208.893,Z 408.945,A -85,B 0,C 180,E1 -21288.832,E2 -21288.832} C_VEL
LIN {X 0,Y 209.118,Z 409.647,A -85,B 0,C 180,E1 -21289.037,E2 -21289.037} C_VEL
LIN {X 0,Y 211.167,Z 413.416,A -85,B 0,C 180,E1 -21289.678,E2 -21289.678} C_VEL
LIN {X 0,Y 212.87,Z 416.365,A -85,B 0,C 180,E1 -21290.189,E2 -21290.189} C_VEL
LIN {X 0,Y 214.023,Z 419.799,A -85,B 0,C 180,E1 -21290.589,E2 -21290.589} C_VEL
LIN {X 0,Y 215.293,Z 427.355,A -85,B 0,C 180,E1 -21291.181,E2 -21291.181} C_VEL
LIN {X 0,Y 216.676,Z 437.098,A -85,B 0,C 180,E1 -21291.874,E2 -21291.874} C_VEL
LIN {X 0,Y 218.494,Z 442.401,A -85,B 0,C 180,E1 -21292.459,E2 -21292.459} C_VEL
LIN {X 0,Y 222.225,Z 451.787,A -85,B 0,C 180,E1 -21293.557,E2 -21293.557} C_VEL
LIN {X 0,Y 224.34,Z 469.32,A -85,B 0,C 180,E1 -21294.626,E2 -21294.626} C_VEL
LIN {X 0,Y 222.07,Z 518.977,A -85,B 0,C 180,E1 -21296.196,E2 -21296.196} C_VEL
LIN {X 0,Y 220.473,Z 532.697,A -85,B 0,C 180,E1 -21296.947,E2 -21296.947} C_VEL
LIN {X 0,Y 218.496,Z 544.762,A -85,B 0,C 180,E1 -21297.946,E2 -21297.946} C_VEL
LIN {X 0,Y 215.844,Z 557.437,A -85,B 0,C 180,E1 -21299.42,E2 -21299.42} C_VEL
LIN {X 0,Y 213.038,Z 568.715,A -85,B 0,C 180,E1 -21301.154,E2 -21301.154} C_VEL
LIN {X 0,Y 210.113,Z 578.877,A -85,B 0,C 180,E1 -21303.157,E2 -21303.157} C_VEL
LIN {X 0,Y 207.198,Z 588.035,A -85,B 0,C 180,E1 -21305.449,E2 -21305.449} C_VEL
LIN {X 0,Y 204.576,Z 596.28,A -85,B 0,C 180,E1 -21308.057,E2 -21308.057} C_VEL
LIN {X 0,Y 202.81,Z 601.934,A -85,B 0,C 180,E1 -21310.253,E2 -21310.253} C_VEL
LIN {X 0,Y 201.041,Z 607.211,A -85,B 0,C 180,E1 -21312.714,E2 -21312.714} C_VEL
LIN {X 0,Y 199.274,Z 612.325,A -85,B 0,C 180,E1 -21315.708,E2 -21315.708} C_VEL
LIN {X 0,Y 198.209,Z 616.309,A -85,B 0,C 180,E1 -21318.755,E2 -21318.755} C_VEL
LIN {X 0,Y 197.577,Z 619.258,A -85,B 0,C 180,E1 -21321.82,E2 -21321.82} C_VEL
LIN {X 0,Y 197.341,Z 620.662,A -85,B 0,C 180,E1 -21323.867,E2 -21323.867} C_VEL
LIN {X 0,Y 197.313,Z 622.283,A -85,B 0,C 180,E1 -21327.959,E2 -21327.959} C_VEL
LIN {X 0,Y 197.469,Z 622.502,A -85,B 0,C 180,E1 -21330,E2 -21330} C_VEL
LIN {X 0,Y 197.317,Z 622.271,A -85,B 0,C 180,E1 -21332.041,E2 -21332.041} C_VEL
LIN {X 0,Y 197.286,Z 621.649,A -85,B 0,C 180,E1 -21334.086,E2 -21334.086} C_VEL
LIN {X 0,Y 197.338,Z 620.635,A -85,B 0,C 180,E1 -21336.133,E2 -21336.133} C_VEL
LIN {X 0,Y 197.565,Z 619.218,A -85,B 0,C 180,E1 -21338.18,E2 -21338.18} C_VEL
LIN {X 0,Y 198.208,Z 616.252,A -85,B 0,C 180,E1 -21341.245,E2 -21341.245} C_VEL
LIN {X 0,Y 199.271,Z 612.246,A -85,B 0,C 180,E1 -21344.293,E2 -21344.293} C_VEL
LIN {X 0,Y 201.397,Z 606.107,A -85,B 0,C 180,E1 -21347.778,E2 -21347.778} C_VEL
LIN {X 0,Y 203.613,Z 599.542,A -85,B 0,C 180,E1 -21350.661,E2 -21350.661} C_VEL
LIN {X 0,Y 206.244,Z 591.091,A -85,B 0,C 180,E1 -21353.602,E2 -21353.602} C_VEL
LIN {X 0,Y 208.933,Z 582.575,A -85,B 0,C 180,E1 -21355.93,E2 -21355.93} C_VEL
LIN {X 0,Y 212.048,Z 572.061,A -85,B 0,C 180,E1 -21358.183,E2 -21358.183} C_VEL
LIN {X 0,Y 215.132,Z 560.228,A -85,B 0,C 180,E1 -21360.15,E2 -21360.15} C_VEL
LIN {X 0,Y 217.712,Z 548.305,A -85,B 0,C 180,E1 -21361.638,E2 -21361.638} C_VEL
LIN {X 0,Y 219.879,Z 535.896,A -85,B 0,C 180,E1 -21362.776,E2 -21362.776} C_VEL
LIN {X 0,Y 221.512,Z 523.312,A -85,B 0,C 180,E1 -21363.574,E2 -21363.574} C_VEL
LIN {X 0,Y 222.508,Z 509.304,A -85,B 0,C 180,E1 -21364.107,E2 -21364.107} C_VEL
LIN {X 0,Y 224.215,Z 468.476,A -85,B 0,C 180,E1 -21365.366,E2 -21365.366} C_VEL
LIN {X 0,Y 221.855,Z 450.744,A -85,B 0,C 180,E1 -21366.489,E2 -21366.489} C_VEL
LIN {X 0,Y 215.876,Z 436.508,A -85,B 0,C 180,E1 -21368.246,E2 -21368.246} C_VEL
LIN {X 0,Y 209.436,Z 423.022,A -85,B 0,C 180,E1 -21370.222,E2 -21370.222} C_VEL
LIN {X 0,Y 203.958,Z 413.226,A -85,B 0,C 180,E1 -21371.973,E2 -21371.973} C_VEL
LIN {X 0,Y 201.642,Z 408.818,A -85,B 0,C 180,E1 -21372.792,E2 -21372.792} C_VEL
LIN {X 0,Y 199.69,Z 401.602,A -85,B 0,C 180,E1 -21377.358,E2 -21377.358} C_VEL
LIN {X 0,Y 199.678,Z 401.612,A -85,B 0,C 180,E1 -21380.742,E2 -21380.742} C_VEL
LIN {X 0,Y 199.632,Z 401.613,A -85,B 0,C 180,E1 -21385.717,E2 -21385.717} C_VEL
LIN {X 0,Y 199.701,Z 401.606,A -85,B 0,C 180,E1 -21388.137,E2 -21388.137} C_VEL
LIN {X 0,Y 199.684,Z 401.604,A -85,B 0,C 180,E1 -21392.771,E2 -21392.771} C_VEL
LIN {X 0,Y 199.734,Z 401.589,A -85,B 0,C 180,E1 -21397.229,E2 -21397.229} C_VEL
LIN {X 0,Y 199.793,Z 401.586,A -85,B 0,C 180,E1 -21401.758,E2 -21401.758} C_VEL
LIN {X 0,Y 199.831,Z 401.593,A -85,B 0,C 180,E1 -21405.748,E2 -21405.748} C_VEL
LIN {X 0,Y 200.067,Z 401.545,A -85,B 0,C 180,E1 -21409.884,E2 -21409.884} C_VEL
LIN {X 0,Y 200.031,Z 401.567,A -85,B 0,C 180,E1 -21413.95,E2 -21413.95} C_VEL
LIN {X 0,Y 200.317,Z 401.516,A -85,B 0,C 180,E1 -21417.989,E2 -21417.989} C_VEL
LIN {X 0,Y 200.478,Z 401.511,A -85,B 0,C 180,E1 -21420,E2 -21420} C_VEL
LIN {X 0,Y 200.027,Z 401.551,A -85,B 0,C 180,E1 -21424.03,E2 -21424.03} C_VEL
LIN {X 0,Y 200.115,Z 401.557,A -85,B 0,C 180,E1 -21428.076,E2 -21428.076} C_VEL
LIN {X 0,Y 199.882,Z 401.567,A -85,B 0,C 180,E1 -21432.179,E2 -21432.179} C_VEL
LIN {X 0,Y 199.8,Z 401.598,A -85,B 0,C 180,E1 -21436.344,E2 -21436.344} C_VEL
LIN {X 0,Y 199.696,Z 401.596,A -85,B 0,C 180,E1 -21440.606,E2 -21440.606} C_VEL
LIN {X 0,Y 199.67,Z 401.601,A -85,B 0,C 180,E1 -21444.985,E2 -21444.985} C_VEL
LIN {X 0,Y 199.672,Z 401.612,A -85,B 0,C 180,E1 -21449.523,E2 -21449.523} C_VEL
LIN {X 0,Y 199.662,Z 401.602,A -85,B 0,C 180,E1 -21452.353,E2 -21452.353} C_VEL
LIN {X 0,Y 199.651,Z 401.606,A -85,B 0,C 180,E1 -21456.757,E2 -21456.757} C_VEL
LIN {X 0,Y 199.677,Z 401.612,A -85,B 0,C 180,E1 -21459.312,E2 -21459.312} C_VEL
LIN {X 0,Y 199.661,Z 401.611,A -85,B 0,C 180,E1 -21462.339,E2 -21462.339} C_VEL
LIN {X 0,Y 199.632,Z 401.726,A -85,B 0,C 180,E1 -21466.931,E2 -21466.931} C_VEL
LIN {X 0,Y 200.547,Z 404.363,A -85,B 0,C 180,E1 -21467.304,E2 -21467.304} C_VEL
LIN {X 0,Y 202.602,Z 406.83,A -85,B 0,C 180,E1 -21467.959,E2 -21467.959} C_VEL
LIN {X 0,Y 204.792,Z 410.243,A -85,B 0,C 180,E1 -21468.672,E2 -21468.672} C_VEL
LIN {X 0,Y 212.392,Z 422.166,A -85,B 0,C 180,E1 -21470.981,E2 -21470.981} C_VEL
LIN {X 0,Y 218.075,Z 432.543,A -85,B 0,C 180,E1 -21472.617,E2 -21472.617} C_VEL
LIN {X 0,Y 224.053,Z 446.007,A -85,B 0,C 180,E1 -21474.312,E2 -21474.312} C_VEL
LIN {X 0,Y 225.189,Z 449.419,A -85,B 0,C 180,E1 -21474.653,E2 -21474.653} C_VEL
LIN {X 0,Y 222.564,Z 503.985,A -85,B 0,C 180,E1 -21476.323,E2 -21476.323} C_VEL
LIN {X 0,Y 221.264,Z 517.278,A -85,B 0,C 180,E1 -21477.055,E2 -21477.055} C_VEL
LIN {X 0,Y 219.564,Z 529.912,A -85,B 0,C 180,E1 -21478.121,E2 -21478.121} C_VEL
LIN {X 0,Y 217.492,Z 541.202,A -85,B 0,C 180,E1 -21479.407,E2 -21479.407} C_VEL
LIN {X 0,Y 214.778,Z 552.823,A -85,B 0,C 180,E1 -21481.142,E2 -21481.142} C_VEL
LIN {X 0,Y 211.978,Z 563.572,A -85,B 0,C 180,E1 -21483.226,E2 -21483.226} C_VEL
LIN {X 0,Y 209.547,Z 572.107,A -85,B 0,C 180,E1 -21485.315,E2 -21485.315} C_VEL
LIN {X 0,Y 206.623,Z 581.003,A -85,B 0,C 180,E1 -21488.029,E2 -21488.029} C_VEL
LIN {X 0,Y 203.984,Z 588.398,A -85,B 0,C 180,E1 -21490.895,E2 -21490.895} C_VEL
LIN {X 0,Y 201.849,Z 594.327,A -85,B 0,C 180,E1 -21493.827,E2 -21493.827} C_VEL
LIN {X 0,Y 200.187,Z 599.008,A -85,B 0,C 180,E1 -21496.809,E2 -21496.809} C_VEL
LIN {X 0,Y 198.917,Z 602.589,A -85,B 0,C 180,E1 -21499.825,E2 -21499.825} C_VEL
LIN {X 0,Y 198.377,Z 604.434,A -85,B 0,C 180,E1 -21501.853,E2 -21501.853} C_VEL
LIN {X 0,Y 197.951,Z 605.821,A -85,B 0,C 180,E1 -21503.886,E2 -21503.886} C_VEL
LIN {X 0,Y 197.539,Z 607.411,A -85,B 0,C 180,E1 -21507.961,E2 -21507.961} C_VEL
LIN {X 0,Y 197.495,Z 607.639,A -85,B 0,C 180,E1 -21510,E2 -21510} C_VEL
LIN {X 0,Y 197.538,Z 607.445,A -85,B 0,C 180,E1 -21512.039,E2 -21512.039} C_VEL
LIN {X 0,Y 197.98,Z 605.896,A -85,B 0,C 180,E1 -21516.113,E2 -21516.113} C_VEL
LIN {X 0,Y 198.381,Z 604.543,A -85,B 0,C 180,E1 -21518.146,E2 -21518.146} C_VEL
LIN {X 0,Y 199.287,Z 601.683,A -85,B 0,C 180,E1 -21521.184,E2 -21521.184} C_VEL
LIN {X 0,Y 200.664,Z 597.799,A -85,B 0,C 180,E1 -21524.191,E2 -21524.191} C_VEL
LIN {X 0,Y 202.471,Z 592.787,A -85,B 0,C 180,E1 -21527.16,E2 -21527.16} C_VEL
LIN {X 0,Y 204.685,Z 586.472,A -85,B 0,C 180,E1 -21530.081,E2 -21530.081} C_VEL
LIN {X 0,Y 207.538,Z 578.56,A -85,B 0,C 180,E1 -21532.919,E2 -21532.919} C_VEL
LIN {X 0,Y 209.883,Z 571.099,A -85,B 0,C 180,E1 -21535.093,E2 -21535.093} C_VEL
LIN {X 0,Y 212.479,Z 561.728,A -85,B 0,C 180,E1 -21537.318,E2 -21537.318} C_VEL
LIN {X 0,Y 215.327,Z 550.967,A -85,B 0,C 180,E1 -21539.312,E2 -21539.312} C_VEL
LIN {X 0,Y 217.754,Z 540.456,A -85,B 0,C 180,E1 -21540.821,E2 -21540.821} C_VEL
LIN {X 0,Y 220.007,Z 527.8,A -85,B 0,C 180,E1 -21542.212,E2 -21542.212} C_VEL
LIN {X 0,Y 221.713,Z 514.895,A -85,B 0,C 180,E1 -21543.233,E2 -21543.233} C_VEL
LIN {X 0,Y 222.83,Z 501.526,A -85,B 0,C 180,E1 -21543.901,E2 -21543.901} C_VEL
LIN {X 0,Y 225.229,Z 449.581,A -85,B 0,C 180,E1 -21545.486,E2 -21545.486} C_VEL
LIN {X 0,Y 224.513,Z 447.082,A -85,B 0,C 180,E1 -21545.715,E2 -21545.715} C_VEL
LIN {X 0,Y 218.982,Z 434.305,A -85,B 0,C 180,E1 -21547.287,E2 -21547.287} C_VEL
LIN {X 0,Y 214.867,Z 426.4,A -85,B 0,C 180,E1 -21548.466,E2 -21548.466} C_VEL
LIN {X 0,Y 209.084,Z 416.872,A -85,B 0,C 180,E1 -21550.167,E2 -21550.167} C_VEL
LIN {X 0,Y 204.507,Z 409.908,A -85,B 0,C 180,E1 -21551.588,E2 -21551.588} C_VEL
LIN {X 0,Y 202.161,Z 406.246,A -85,B 0,C 180,E1 -21552.359,E2 -21552.359} C_VEL
LIN {X 0,Y 200.327,Z 403.916,A -85,B 0,C 180,E1 -21552.956,E2 -21552.956} C_VEL
LIN {X 0,Y 199.607,Z 401.618,A -85,B 0,C 180,E1 -21553.306,E2 -21553.306} C_VEL
LIN {X 0,Y 199.655,Z 401.592,A -85,B 0,C 180,E1 -21558.024,E2 -21558.024} C_VEL
LIN {X 0,Y 199.679,Z 401.613,A -85,B 0,C 180,E1 -21560.742,E2 -21560.742} C_VEL
LIN {X 0,Y 199.633,Z 401.613,A -85,B 0,C 180,E1 -21565.717,E2 -21565.717} C_VEL
LIN {X 0,Y 199.702,Z 401.607,A -85,B 0,C 180,E1 -21568.137,E2 -21568.137} C_VEL
LIN {X 0,Y 199.685,Z 401.607,A -85,B 0,C 180,E1 -21572.771,E2 -21572.771} C_VEL
LIN {X 0,Y 199.735,Z 401.594,A -85,B 0,C 180,E1 -21577.229,E2 -21577.229} C_VEL
LIN {X 0,Y 199.793,Z 401.587,A -85,B 0,C 180,E1 -21581.757,E2 -21581.757} C_VEL
LIN {X 0,Y 199.832,Z 401.593,A -85,B 0,C 180,E1 -21585.748,E2 -21585.748} C_VEL
LIN {X 0,Y 200.067,Z 401.553,A -85,B 0,C 180,E1 -21589.884,E2 -21589.884} C_VEL
LIN {X 0,Y 200.03,Z 401.562,A -85,B 0,C 180,E1 -21593.949,E2 -21593.949} C_VEL
LIN {X 0,Y 200.318,Z 401.532,A -85,B 0,C 180,E1 -21597.989,E2 -21597.989} C_VEL
LIN {X 0,Y 200.478,Z 401.509,A -85,B 0,C 180,E1 -21600,E2 -21600} C_VEL
LIN {X 0,Y 200.028,Z 401.565,A -85,B 0,C 180,E1 -21604.029,E2 -21604.029} C_VEL
LIN {X 0,Y 200.107,Z 401.544,A -85,B 0,C 180,E1 -21608.076,E2 -21608.076} C_VEL
LIN {X 0,Y 199.91,Z 401.582,A -85,B 0,C 180,E1 -21612.177,E2 -21612.177} C_VEL
LIN {X 0,Y 199.801,Z 401.594,A -85,B 0,C 180,E1 -21616.344,E2 -21616.344} C_VEL
LIN {X 0,Y 199.696,Z 401.601,A -85,B 0,C 180,E1 -21620.606,E2 -21620.606} C_VEL
LIN {X 0,Y 199.67,Z 401.605,A -85,B 0,C 180,E1 -21624.985,E2 -21624.985} C_VEL
LIN {X 0,Y 199.672,Z 401.611,A -85,B 0,C 180,E1 -21629.523,E2 -21629.523} C_VEL
LIN {X 0,Y 199.661,Z 401.607,A -85,B 0,C 180,E1 -21632.353,E2 -21632.353} C_VEL
LIN {X 0,Y 199.651,Z 401.605,A -85,B 0,C 180,E1 -21636.757,E2 -21636.757} C_VEL
LIN {X 0,Y 199.677,Z 401.608,A -85,B 0,C 180,E1 -21639.312,E2 -21639.312} C_VEL
LIN {X 0,Y 199.7,Z 401.679,A -85,B 0,C 180,E1 -21642.639,E2 -21642.639} C_VEL
LIN {X 0,Y 201.616,Z 408.859,A -85,B 0,C 180,E1 -21647.138,E2 -21647.138} C_VEL
LIN {X 0,Y 204.127,Z 413.43,A -85,B 0,C 180,E1 -21647.995,E2 -21647.995} C_VEL
LIN {X 0,Y 208.432,Z 421.315,A -85,B 0,C 180,E1 -21649.393,E2 -21649.393} C_VEL
LIN {X 0,Y 213.492,Z 431.234,A -85,B 0,C 180,E1 -21650.958,E2 -21650.958} C_VEL
LIN {X 0,Y 218.494,Z 442.401,A -85,B 0,C 180,E1 -21652.459,E2 -21652.459} C_VEL
LIN {X 0,Y 219.725,Z 445.803,A -85,B 0,C 180,E1 -21652.839,E2 -21652.839} C_VEL
LIN {X 0,Y 220.437,Z 451.488,A -85,B 0,C 180,E1 -21653.204,E2 -21653.204} C_VEL
LIN {X 0,Y 220.201,Z 457.408,A -85,B 0,C 180,E1 -21653.394,E2 -21653.394} C_VEL
LIN {X 0,Y 218.392,Z 473.915,A -85,B 0,C 180,E1 -21653.704,E2 -21653.704} C_VEL
LIN {X 0,Y 216.229,Z 518.524,A -85,B 0,C 180,E1 -21655.141,E2 -21655.141} C_VEL
LIN {X 0,Y 214.642,Z 531.888,A -85,B 0,C 180,E1 -21655.877,E2 -21655.877} C_VEL
LIN {X 0,Y 212.525,Z 544.502,A -85,B 0,C 180,E1 -21656.933,E2 -21656.933} C_VEL
LIN {X 0,Y 209.758,Z 557.175,A -85,B 0,C 180,E1 -21658.432,E2 -21658.432} C_VEL
LIN {X 0,Y 206.852,Z 568.452,A -85,B 0,C 180,E1 -21660.206,E2 -21660.206} C_VEL
LIN {X 0,Y 203.773,Z 578.611,A -85,B 0,C 180,E1 -21662.251,E2 -21662.251} C_VEL
LIN {X 0,Y 200.735,Z 587.769,A -85,B 0,C 180,E1 -21664.604,E2 -21664.604} C_VEL
LIN {X 0,Y 197.763,Z 596.642,A -85,B 0,C 180,E1 -21667.514,E2 -21667.514} C_VEL
LIN {X 0,Y 195.684,Z 602.79,A -85,B 0,C 180,E1 -21670.051,E2 -21670.051} C_VEL
LIN {X 0,Y 193.541,Z 608.768,A -85,B 0,C 180,E1 -21673.112,E2 -21673.112} C_VEL
LIN {X 0,Y 191.939,Z 613.498,A -85,B 0,C 180,E1 -21676.232,E2 -21676.232} C_VEL
LIN {X 0,Y 190.956,Z 617.121,A -85,B 0,C 180,E1 -21679.396,E2 -21679.396} C_VEL
LIN {X 0,Y 190.524,Z 618.99,A -85,B 0,C 180,E1 -21681.515,E2 -21681.515} C_VEL
LIN {X 0,Y 190.278,Z 620.395,A -85,B 0,C 180,E1 -21683.638,E2 -21683.638} C_VEL
LIN {X 0,Y 190.17,Z 621.577,A -85,B 0,C 180,E1 -21686.22,E2 -21686.22} C_VEL
LIN {X 0,Y 190.385,Z 622.235,A -85,B 0,C 180,E1 -21690,E2 -21690} C_VEL
LIN {X 0,Y 190.179,Z 621.542,A -85,B 0,C 180,E1 -21693.82,E2 -21693.82} C_VEL
LIN {X 0,Y 190.275,Z 620.367,A -85,B 0,C 180,E1 -21696.362,E2 -21696.362} C_VEL
LIN {X 0,Y 190.515,Z 618.949,A -85,B 0,C 180,E1 -21698.485,E2 -21698.485} C_VEL
LIN {X 0,Y 191.223,Z 615.983,A -85,B 0,C 180,E1 -21701.662,E2 -21701.662} C_VEL
LIN {X 0,Y 192.358,Z 611.977,A -85,B 0,C 180,E1 -21704.818,E2 -21704.818} C_VEL
LIN {X 0,Y 194.612,Z 605.837,A -85,B 0,C 180,E1 -21708.42,E2 -21708.42} C_VEL
LIN {X 0,Y 197.14,Z 598.761,A -85,B 0,C 180,E1 -21711.598,E2 -21711.598} C_VEL
LIN {X 0,Y 199.71,Z 590.82,A -85,B 0,C 180,E1 -21714.424,E2 -21714.424} C_VEL
LIN {X 0,Y 202.546,Z 582.304,A -85,B 0,C 180,E1 -21716.812,E2 -21716.812} C_VEL
LIN {X 0,Y 205.786,Z 571.789,A -85,B 0,C 180,E1 -21719.121,E2 -21719.121} C_VEL
LIN {X 0,Y 209.02,Z 559.956,A -85,B 0,C 180,E1 -21721.128,E2 -21721.128} C_VEL
LIN {X 0,Y 211.694,Z 548.031,A -85,B 0,C 180,E1 -21722.647,E2 -21722.647} C_VEL
LIN {X 0,Y 213.944,Z 535.621,A -85,B 0,C 180,E1 -21723.806,E2 -21723.806} C_VEL
LIN {X 0,Y 215.655,Z 522.767,A -85,B 0,C 180,E1 -21724.632,E2 -21724.632} C_VEL
LIN {X 0,Y 216.725,Z 507.801,A -85,B 0,C 180,E1 -21725.197,E2 -21725.197} C_VEL
LIN {X 0,Y 218.356,Z 469.228,A -85,B 0,C 180,E1 -21726.423,E2 -21726.423} C_VEL
LIN {X 0,Y 216.349,Z 453.437,A -85,B 0,C 180,E1 -21727.454,E2 -21727.454} C_VEL
LIN {X 0,Y 209.919,Z 438.135,A -85,B 0,C 180,E1 -21729.455,E2 -21729.455} C_VEL
LIN {X 0,Y 204.26,Z 426.372,A -85,B 0,C 180,E1 -21731.295,E2 -21731.295} C_VEL
LIN {X 0,Y 199.463,Z 417.679,A -85,B 0,C 180,E1 -21732.92,E2 -21732.92} C_VEL
LIN {X 0,Y 196.681,Z 412.814,A -85,B 0,C 180,E1 -21733.91,E2 -21733.91} C_VEL
LIN {X 0,Y 194.272,Z 408.405,A -85,B 0,C 180,E1 -21734.861,E2 -21734.861} C_VEL
LIN {X 0,Y 192.585,Z 402.489,A -85,B 0,C 180,E1 -21738.938,E2 -21738.938} C_VEL
LIN {X 0,Y 192.617,Z 402.485,A -85,B 0,C 180,E1 -21743.388,E2 -21743.388} C_VEL
LIN {X 0,Y 192.605,Z 402.483,A -85,B 0,C 180,E1 -21747.059,E2 -21747.059} C_VEL
LIN {X 0,Y 192.662,Z 402.472,A -85,B 0,C 180,E1 -21751.691,E2 -21751.691} C_VEL
LIN {X 0,Y 192.703,Z 402.464,A -85,B 0,C 180,E1 -21756.348,E2 -21756.348} C_VEL
LIN {X 0,Y 192.729,Z 402.467,A -85,B 0,C 180,E1 -21761.457,E2 -21761.457} C_VEL
LIN {X 0,Y 192.759,Z 402.47,A -85,B 0,C 180,E1 -21765.213,E2 -21765.213} C_VEL
LIN {X 0,Y 192.978,Z 402.427,A -85,B 0,C 180,E1 -21769.508,E2 -21769.508} C_VEL
LIN {X 0,Y 193.058,Z 402.428,A -85,B 0,C 180,E1 -21771.627,E2 -21771.627} C_VEL
LIN {X 0,Y 193.259,Z 402.393,A -85,B 0,C 180,E1 -21777.916,E2 -21777.916} C_VEL
LIN {X 0,Y 193.442,Z 402.387,A -85,B 0,C 180,E1 -21780,E2 -21780} C_VEL
LIN {X 0,Y 192.973,Z 402.428,A -85,B 0,C 180,E1 -21784.177,E2 -21784.177} C_VEL
LIN {X 0,Y 193.064,Z 402.436,A -85,B 0,C 180,E1 -21788.373,E2 -21788.373} C_VEL
LIN {X 0,Y 192.806,Z 402.448,A -85,B 0,C 180,E1 -21792.633,E2 -21792.633} C_VEL
LIN {X 0,Y 192.754,Z 402.472,A -85,B 0,C 180,E1 -21796.959,E2 -21796.959} C_VEL
LIN {X 0,Y 192.633,Z 402.483,A -85,B 0,C 180,E1 -21801.398,E2 -21801.398} C_VEL
LIN {X 0,Y 192.661,Z 402.48,A -85,B 0,C 180,E1 -21804.225,E2 -21804.225} C_VEL
LIN {X 0,Y 192.648,Z 402.489,A -85,B 0,C 180,E1 -21808.893,E2 -21808.893} C_VEL
LIN {X 0,Y 192.598,Z 402.488,A -85,B 0,C 180,E1 -21813.186,E2 -21813.186} C_VEL
LIN {X 0,Y 192.599,Z 402.492,A -85,B 0,C 180,E1 -21818.341,E2 -21818.341} C_VEL
LIN {X 0,Y 192.599,Z 402.495,A -85,B 0,C 180,E1 -21823.131,E2 -21823.131} C_VEL
LIN {X 0,Y 192.596,Z 402.524,A -85,B 0,C 180,E1 -21824.962,E2 -21824.962} C_VEL
LIN {X 0,Y 193.53,Z 405.256,A -85,B 0,C 180,E1 -21825.382,E2 -21825.382} C_VEL
LIN {X 0,Y 195.822,Z 408.104,A -85,B 0,C 180,E1 -21826.189,E2 -21826.189} C_VEL
LIN {X 0,Y 198.021,Z 411.371,A -85,B 0,C 180,E1 -21826.962,E2 -21826.962} C_VEL
LIN {X 0,Y 205.691,Z 423.101,A -85,B 0,C 180,E1 -21829.477,E2 -21829.477} C_VEL
LIN {X 0,Y 212.666,Z 435.383,A -85,B 0,C 180,E1 -21831.603,E2 -21831.603} C_VEL
LIN {X 0,Y 218.958,Z 449.822,A -85,B 0,C 180,E1 -21833.492,E2 -21833.492} C_VEL
LIN {X 0,Y 219.385,Z 451.509,A -85,B 0,C 180,E1 -21833.642,E2 -21833.642} C_VEL
LIN {X 0,Y 216.626,Z 505.094,A -85,B 0,C 180,E1 -21835.321,E2 -21835.321} C_VEL
LIN {X 0,Y 215.163,Z 518.815,A -85,B 0,C 180,E1 -21836.113,E2 -21836.113} C_VEL
LIN {X 0,Y 213.375,Z 531.27,A -85,B 0,C 180,E1 -21837.221,E2 -21837.221} C_VEL
LIN {X 0,Y 211.068,Z 543.054,A -85,B 0,C 180,E1 -21838.65,E2 -21838.65} C_VEL
LIN {X 0,Y 208.261,Z 554.38,A -85,B 0,C 180,E1 -21840.427,E2 -21840.427} C_VEL
LIN {X 0,Y 205.666,Z 563.843,A -85,B 0,C 180,E1 -21842.335,E2 -21842.335} C_VEL
LIN {X 0,Y 203.026,Z 572.672,A -85,B 0,C 180,E1 -21844.558,E2 -21844.558} C_VEL
LIN {X 0,Y 200.066,Z 581.272,A -85,B 0,C 180,E1 -21847.269,E2 -21847.269} C_VEL
LIN {X 0,Y 197.291,Z 588.667,A -85,B 0,C 180,E1 -21850.22,E2 -21850.22} C_VEL
LIN {X 0,Y 195.045,Z 594.595,A -85,B 0,C 180,E1 -21853.246,E2 -21853.246} C_VEL
LIN {X 0,Y 193.269,Z 599.277,A -85,B 0,C 180,E1 -21856.328,E2 -21856.328} C_VEL
LIN {X 0,Y 191.923,Z 602.857,A -85,B 0,C 180,E1 -21859.45,E2 -21859.45} C_VEL
LIN {X 0,Y 191.354,Z 604.702,A -85,B 0,C 180,E1 -21861.552,E2 -21861.552} C_VEL
LIN {X 0,Y 190.86,Z 606.182,A -85,B 0,C 180,E1 -21863.838,E2 -21863.838} C_VEL
LIN {X 0,Y 190.463,Z 607.678,A -85,B 0,C 180,E1 -21867.885,E2 -21867.885} C_VEL
LIN {X 0,Y 190.416,Z 607.905,A -85,B 0,C 180,E1 -21870,E2 -21870} C_VEL
LIN {X 0,Y 190.463,Z 607.711,A -85,B 0,C 180,E1 -21872.115,E2 -21872.115} C_VEL
LIN {X 0,Y 190.925,Z 606.162,A -85,B 0,C 180,E1 -21876.34,E2 -21876.34} C_VEL
LIN {X 0,Y 191.36,Z 604.809,A -85,B 0,C 180,E1 -21878.447,E2 -21878.447} C_VEL
LIN {X 0,Y 192.32,Z 601.95,A -85,B 0,C 180,E1 -21881.594,E2 -21881.594} C_VEL
LIN {X 0,Y 193.77,Z 598.066,A -85,B 0,C 180,E1 -21884.707,E2 -21884.707} C_VEL
LIN {X 0,Y 195.707,Z 593.053,A -85,B 0,C 180,E1 -21887.772,E2 -21887.772} C_VEL
LIN {X 0,Y 198.045,Z 586.737,A -85,B 0,C 180,E1 -21890.785,E2 -21890.785} C_VEL
LIN {X 0,Y 201.029,Z 578.825,A -85,B 0,C 180,E1 -21893.705,E2 -21893.705} C_VEL
LIN {X 0,Y 203.85,Z 570.004,A -85,B 0,C 180,E1 -21896.313,E2 -21896.313} C_VEL
LIN {X 0,Y 206.844,Z 559.826,A -85,B 0,C 180,E1 -21898.68,E2 -21898.68} C_VEL
LIN {X 0,Y 209.545,Z 549.834,A -85,B 0,C 180,E1 -21900.482,E2 -21900.482} C_VEL
LIN {X 0,Y 212.061,Z 538.957,A -85,B 0,C 180,E1 -21902.022,E2 -21902.022} C_VEL
LIN {X 0,Y 214.219,Z 526.933,A -85,B 0,C 180,E1 -21903.334,E2 -21903.334} C_VEL
LIN {X 0,Y 215.943,Z 514.056,A -85,B 0,C 180,E1 -21904.331,E2 -21904.331} C_VEL
LIN {X 0,Y 217.018,Z 500.597,A -85,B 0,C 180,E1 -21904.994,E2 -21904.994} C_VEL
LIN {X 0,Y 219.411,Z 450.868,A -85,B 0,C 180,E1 -21906.535,E2 -21906.535} C_VEL
LIN {X 0,Y 214.003,Z 438.167,A -85,B 0,C 180,E1 -21908.156,E2 -21908.156} C_VEL
LIN {X 0,Y 209.257,Z 428.999,A -85,B 0,C 180,E1 -21909.594,E2 -21909.594} C_VEL
LIN {X 0,Y 201.003,Z 415.687,A -85,B 0,C 180,E1 -21912.214,E2 -21912.214} C_VEL
LIN {X 0,Y 197.435,Z 410.674,A -85,B 0,C 180,E1 -21913.415,E2 -21913.415} C_VEL
LIN {X 0,Y 195.279,Z 407.241,A -85,B 0,C 180,E1 -21914.195,E2 -21914.195} C_VEL
LIN {X 0,Y 193.344,Z 404.907,A -85,B 0,C 180,E1 -21914.88,E2 -21914.88} C_VEL
LIN {X 0,Y 192.596,Z 402.481,A -85,B 0,C 180,E1 -21915.291,E2 -21915.291} C_VEL
LIN {X 0,Y 192.587,Z 402.493,A -85,B 0,C 180,E1 -21920.025,E2 -21920.025} C_VEL
LIN {X 0,Y 192.6,Z 402.495,A -85,B 0,C 180,E1 -21924.279,E2 -21924.279} C_VEL
LIN {X 0,Y 192.605,Z 402.495,A -85,B 0,C 180,E1 -21929.279,E2 -21929.279} C_VEL
LIN {X 0,Y 192.662,Z 402.476,A -85,B 0,C 180,E1 -21931.691,E2 -21931.691} C_VEL
LIN {X 0,Y 192.703,Z 402.469,A -85,B 0,C 180,E1 -21936.348,E2 -21936.348} C_VEL
LIN {X 0,Y 192.729,Z 402.468,A -85,B 0,C 180,E1 -21941.457,E2 -21941.457} C_VEL
LIN {X 0,Y 192.76,Z 402.473,A -85,B 0,C 180,E1 -21945.213,E2 -21945.213} C_VEL
LIN {X 0,Y 192.978,Z 402.433,A -85,B 0,C 180,E1 -21949.508,E2 -21949.508} C_VEL
LIN {X 0,Y 193.058,Z 402.438,A -85,B 0,C 180,E1 -21951.627,E2 -21951.627} C_VEL
LIN {X 0,Y 193.26,Z 402.411,A -85,B 0,C 180,E1 -21957.916,E2 -21957.916} C_VEL
LIN {X 0,Y 193.442,Z 402.386,A -85,B 0,C 180,E1 -21960,E2 -21960} C_VEL
LIN {X 0,Y 192.975,Z 402.443,A -85,B 0,C 180,E1 -21964.177,E2 -21964.177} C_VEL
LIN {X 0,Y 193.058,Z 402.421,A -85,B 0,C 180,E1 -21968.373,E2 -21968.373} C_VEL
LIN {X 0,Y 192.849,Z 402.457,A -85,B 0,C 180,E1 -21972.63,E2 -21972.63} C_VEL
LIN {X 0,Y 192.754,Z 402.475,A -85,B 0,C 180,E1 -21976.959,E2 -21976.959} C_VEL
LIN {X 0,Y 192.633,Z 402.487,A -85,B 0,C 180,E1 -21981.398,E2 -21981.398} C_VEL
LIN {X 0,Y 192.661,Z 402.478,A -85,B 0,C 180,E1 -21984.225,E2 -21984.225} C_VEL
LIN {X 0,Y 192.647,Z 402.487,A -85,B 0,C 180,E1 -21988.893,E2 -21988.893} C_VEL
LIN {X 0,Y 192.598,Z 402.482,A -85,B 0,C 180,E1 -21993.186,E2 -21993.186} C_VEL
LIN {X 0,Y 192.598,Z 402.488,A -85,B 0,C 180,E1 -21998.341,E2 -21998.341} C_VEL
LIN {X 0,Y 192.585,Z 402.539,A -85,B 0,C 180,E1 -22001.062,E2 -22001.062} C_VEL
LIN {X 0,Y 194.34,Z 408.625,A -85,B 0,C 180,E1 -22005.119,E2 -22005.119} C_VEL
LIN {X 0,Y 196.843,Z 413.062,A -85,B 0,C 180,E1 -22006.054,E2 -22006.054} C_VEL
LIN {X 0,Y 203.069,Z 424.097,A -85,B 0,C 180,E1 -22008.223,E2 -22008.223} C_VEL
LIN {X 0,Y 208.588,Z 435.083,A -85,B 0,C 180,E1 -22010.036,E2 -22010.036} C_VEL
LIN {X 0,Y 215.975,Z 452.264,A -85,B 0,C 180,E1 -22012.353,E2 -22012.353} C_VEL
LIN {X 0,Y 216.778,Z 454.918,A -85,B 0,C 180,E1 -22012.624,E2 -22012.624} C_VEL
LIN {X 0,Y 218.551,Z 470.144,A -85,B 0,C 180,E1 -22013.584,E2 -22013.584} C_VEL
LIN {X 0,Y 218.392,Z 473.915,A -85,B 0,C 180,E1 -22013.704,E2 -22013.704} C_VEL
LIN {X 0,Y 217.637,Z 479.76,A -85,B 0,C 180,E1 -22013.793,E2 -22013.793} C_VEL
LIN {X 0,Y 212.018,Z 498.764,A -85,B 0,C 180,E1 -22013.47,E2 -22013.47} C_VEL
LIN {X 0,Y 211.219,Z 504.612,A -85,B 0,C 180,E1 -22013.552,E2 -22013.552} C_VEL
LIN {X 0,Y 210.165,Z 521.08,A -85,B 0,C 180,E1 -22014.163,E2 -22014.163} C_VEL
LIN {X 0,Y 208.514,Z 533.6,A -85,B 0,C 180,E1 -22014.922,E2 -22014.922} C_VEL
LIN {X 0,Y 206.18,Z 546.241,A -85,B 0,C 180,E1 -22016.072,E2 -22016.072} C_VEL
LIN {X 0,Y 203.348,Z 558.497,A -85,B 0,C 180,E1 -22017.609,E2 -22017.609} C_VEL
LIN {X 0,Y 200.327,Z 569.438,A -85,B 0,C 180,E1 -22019.424,E2 -22019.424} C_VEL
LIN {X 0,Y 196.859,Z 580.305,A -85,B 0,C 180,E1 -22021.769,E2 -22021.769} C_VEL
LIN {X 0,Y 193.746,Z 589.139,A -85,B 0,C 180,E1 -22024.197,E2 -22024.197} C_VEL
LIN {X 0,Y 190.932,Z 597.077,A -85,B 0,C 180,E1 -22026.959,E2 -22026.959} C_VEL
LIN {X 0,Y 188.567,Z 603.64,A -85,B 0,C 180,E1 -22029.834,E2 -22029.834} C_VEL
LIN {X 0,Y 186.742,Z 608.502,A -85,B 0,C 180,E1 -22032.478,E2 -22032.478} C_VEL
LIN {X 0,Y 184.995,Z 613.229,A -85,B 0,C 180,E1 -22035.704,E2 -22035.704} C_VEL
LIN {X 0,Y 183.939,Z 616.852,A -85,B 0,C 180,E1 -22038.987,E2 -22038.987} C_VEL
LIN {X 0,Y 183.492,Z 618.723,A -85,B 0,C 180,E1 -22041.187,E2 -22041.187} C_VEL
LIN {X 0,Y 183.21,Z 620.128,A -85,B 0,C 180,E1 -22043.392,E2 -22043.392} C_VEL
LIN {X 0,Y 183.125,Z 621.749,A -85,B 0,C 180,E1 -22047.801,E2 -22047.801} C_VEL
LIN {X 0,Y 183.284,Z 621.968,A -85,B 0,C 180,E1 -22050,E2 -22050} C_VEL
LIN {X 0,Y 183.09,Z 621.408,A -85,B 0,C 180,E1 -22053.602,E2 -22053.602} C_VEL
LIN {X 0,Y 183.207,Z 620.099,A -85,B 0,C 180,E1 -22056.608,E2 -22056.608} C_VEL
LIN {X 0,Y 183.485,Z 618.681,A -85,B 0,C 180,E1 -22058.813,E2 -22058.813} C_VEL
LIN {X 0,Y 184.258,Z 615.715,A -85,B 0,C 180,E1 -22062.109,E2 -22062.109} C_VEL
LIN {X 0,Y 185.469,Z 611.707,A -85,B 0,C 180,E1 -22065.382,E2 -22065.382} C_VEL
LIN {X 0,Y 187.826,Z 605.566,A -85,B 0,C 180,E1 -22069.111,E2 -22069.111} C_VEL
LIN {X 0,Y 190.418,Z 598.776,A -85,B 0,C 180,E1 -22072.27,E2 -22072.27} C_VEL
LIN {X 0,Y 193.236,Z 590.549,A -85,B 0,C 180,E1 -22075.299,E2 -22075.299} C_VEL
LIN {X 0,Y 196.227,Z 582.033,A -85,B 0,C 180,E1 -22077.749,E2 -22077.749} C_VEL
LIN {X 0,Y 199.582,Z 571.517,A -85,B 0,C 180,E1 -22080.118,E2 -22080.118} C_VEL
LIN {X 0,Y 202.965,Z 559.684,A -85,B 0,C 180,E1 -22082.166,E2 -22082.166} C_VEL
LIN {X 0,Y 205.741,Z 547.757,A -85,B 0,C 180,E1 -22083.716,E2 -22083.716} C_VEL
LIN {X 0,Y 208.096,Z 535.346,A -85,B 0,C 180,E1 -22084.891,E2 -22084.891} C_VEL
LIN {X 0,Y 209.892,Z 522.356,A -85,B 0,C 180,E1 -22085.736,E2 -22085.736} C_VEL
LIN {X 0,Y 210.964,Z 507.472,A -85,B 0,C 180,E1 -22086.31,E2 -22086.31} C_VEL
LIN {X 0,Y 212.646,Z 470.225,A -85,B 0,C 180,E1 -22087.514,E2 -22087.514} C_VEL
LIN {X 0,Y 210.885,Z 456.048,A -85,B 0,C 180,E1 -22088.477,E2 -22088.477} C_VEL
LIN {X 0,Y 204.195,Z 440.091,A -85,B 0,C 180,E1 -22090.688,E2 -22090.688} C_VEL
LIN {X 0,Y 197.876,Z 427.094,A -85,B 0,C 180,E1 -22092.888,E2 -22092.888} C_VEL
LIN {X 0,Y 192.463,Z 417.562,A -85,B 0,C 180,E1 -22094.875,E2 -22094.875} C_VEL
LIN {X 0,Y 189.685,Z 412.89,A -85,B 0,C 180,E1 -22095.956,E2 -22095.956} C_VEL
LIN {X 0,Y 187.013,Z 408.393,A -85,B 0,C 180,E1 -22097.047,E2 -22097.047} C_VEL
LIN {X 0,Y 186.795,Z 407.716,A -85,B 0,C 180,E1 -22097.372,E2 -22097.372} C_VEL
LIN {X 0,Y 185.553,Z 403.369,A -85,B 0,C 180,E1 -22100.623,E2 -22100.623} C_VEL
LIN {X 0,Y 185.519,Z 403.373,A -85,B 0,C 180,E1 -22105.372,E2 -22105.372} C_VEL
LIN {X 0,Y 185.58,Z 403.356,A -85,B 0,C 180,E1 -22110.575,E2 -22110.575} C_VEL
LIN {X 0,Y 185.585,Z 403.356,A -85,B 0,C 180,E1 -22115.382,E2 -22115.382} C_VEL
LIN {X 0,Y 185.672,Z 403.348,A -85,B 0,C 180,E1 -22121.133,E2 -22121.133} C_VEL
LIN {X 0,Y 185.691,Z 403.346,A -85,B 0,C 180,E1 -22124.637,E2 -22124.637} C_VEL
LIN {X 0,Y 185.921,Z 403.306,A -85,B 0,C 180,E1 -22129.359,E2 -22129.359} C_VEL
LIN {X 0,Y 185.957,Z 403.322,A -85,B 0,C 180,E1 -22133.49,E2 -22133.49} C_VEL
LIN {X 0,Y 186.204,Z 403.271,A -85,B 0,C 180,E1 -22137.837,E2 -22137.837} C_VEL
LIN {X 0,Y 186.405,Z 403.264,A -85,B 0,C 180,E1 -22140,E2 -22140} C_VEL
